LIN {X 0,Y 360.021,Z 1147.139,A -85,B 0,C 180,E1 17549.045,E2 17549.045} C_VEL
LIN {X 0,Y 360.007,Z 1146.189,A -85,B 0,C 180,E1 17546.018,E2 17546.018} C_VEL
LIN {X 0,Y 360.001,Z 1143.714,A -85,B 0,C 180,E1 17542.339,E2 17542.339} C_VEL
LIN {X 0,Y 360.288,Z 1139.777,A -85,B 0,C 180,E1 17538.798,E2 17538.798} C_VEL
LIN {X 0,Y 360.939,Z 1135.011,A -85,B 0,C 180,E1 17535.563,E2 17535.563} C_VEL
LIN {X 0,Y 362.46,Z 1127.574,A -85,B 0,C 180,E1 17531.617,E2 17531.617} C_VEL
LIN {X 0,Y 364.535,Z 1119.65,A -85,B 0,C 180,E1 17528.266,E2 17528.266} C_VEL
LIN {X 0,Y 367.67,Z 1109.706,A -85,B 0,C 180,E1 17524.725,E2 17524.725} C_VEL
LIN {X 0,Y 371.821,Z 1097.742,A -85,B 0,C 180,E1 17521.225,E2 17521.225} C_VEL
LIN {X 0,Y 376.526,Z 1085.225,A -85,B 0,C 180,E1 17518.099,E2 17518.099} C_VEL
LIN {X 0,Y 382.373,Z 1070.124,A -85,B 0,C 180,E1 17514.934,E2 17514.934} C_VEL
LIN {X 0,Y 388.351,Z 1054.921,A -85,B 0,C 180,E1 17512.209,E2 17512.209} C_VEL
LIN {X 0,Y 395.187,Z 1037.236,A -85,B 0,C 180,E1 17509.534,E2 17509.534} C_VEL
LIN {X 0,Y 401.308,Z 1020.991,A -85,B 0,C 180,E1 17507.432,E2 17507.432} C_VEL
LIN {X 0,Y 408.852,Z 999.928,A -85,B 0,C 180,E1 17505.125,E2 17505.125} C_VEL
LIN {X 0,Y 414.782,Z 982.18,A -85,B 0,C 180,E1 17503.481,E2 17503.481} C_VEL
LIN {X 0,Y 421.323,Z 961.181,A -85,B 0,C 180,E1 17501.824,E2 17501.824} C_VEL
LIN {X 0,Y 427.122,Z 940.304,A -85,B 0,C 180,E1 17500.463,E2 17500.463} C_VEL
LIN {X 0,Y 432.626,Z 918.319,A -85,B 0,C 180,E1 17499.262,E2 17499.262} C_VEL
LIN {X 0,Y 437.401,Z 895.765,A -85,B 0,C 180,E1 17498.28,E2 17498.28} C_VEL
LIN {X 0,Y 441.245,Z 874.481,A -85,B 0,C 180,E1 17497.536,E2 17497.536} C_VEL
LIN {X 0,Y 444.909,Z 848.294,A -85,B 0,C 180,E1 17496.842,E2 17496.842} C_VEL
LIN {X 0,Y 446.964,Z 825.929,A -85,B 0,C 180,E1 17496.396,E2 17496.396} C_VEL
LIN {X 0,Y 460.098,Z 603.079,A -85,B 0,C 180,E1 17492.792,E2 17492.792} C_VEL
LIN {X 0,Y 461.524,Z 577.948,A -85,B 0,C 180,E1 17492.371,E2 17492.371} C_VEL
LIN {X 0,Y 452.704,Z 561.651,A -85,B 0,C 180,E1 17490.201,E2 17490.201} C_VEL
LIN {X 0,Y 443.998,Z 546.554,A -85,B 0,C 180,E1 17487.859,E2 17487.859} C_VEL
LIN {X 0,Y 434.702,Z 531.507,A -85,B 0,C 180,E1 17485.075,E2 17485.075} C_VEL
LIN {X 0,Y 426.121,Z 518.593,A -85,B 0,C 180,E1 17482.16,E2 17482.16} C_VEL
LIN {X 0,Y 420.35,Z 510.714,A -85,B 0,C 180,E1 17479.959,E2 17479.959} C_VEL
LIN {X 0,Y 416.022,Z 505.286,A -85,B 0,C 180,E1 17478.135,E2 17478.135} C_VEL
LIN {X 0,Y 412.343,Z 500.609,A -85,B 0,C 180,E1 17476.41,E2 17476.41} C_VEL
LIN {X 0,Y 408.2,Z 495.981,A -85,B 0,C 180,E1 17474.251,E2 17474.251} C_VEL
LIN {X 0,Y 406.955,Z 494.027,A -85,B 0,C 180,E1 17473.498,E2 17473.498} C_VEL
LIN {X 0,Y 403.56,Z 490.738,A -85,B 0,C 180,E1 17471.36,E2 17471.36} C_VEL
LIN {X 0,Y 402.048,Z 488.022,A -85,B 0,C 180,E1 17470.17,E2 17470.17} C_VEL
LIN {X 0,Y 398.584,Z 485.25,A -85,B 0,C 180,E1 17467.206,E2 17467.206} C_VEL
LIN {X 0,Y 396.721,Z 481.774,A -85,B 0,C 180,E1 17464.771,E2 17464.771} C_VEL
LIN {X 0,Y 394.33,Z 480.47,A -85,B 0,C 180,E1 17458.838,E2 17458.838} C_VEL
LIN {X 0,Y 395.914,Z 481.333,A -85,B 0,C 180,E1 17452.891,E2 17452.891} C_VEL
LIN {X 0,Y 397.035,Z 482.238,A -85,B 0,C 180,E1 17451.236,E2 17451.236} C_VEL
LIN {X 0,Y 398.95,Z 485.758,A -85,B 0,C 180,E1 17448.873,E2 17448.873} C_VEL
LIN {X 0,Y 402.253,Z 488.401,A -85,B 0,C 180,E1 17446.121,E2 17446.121} C_VEL
LIN {X 0,Y 404.933,Z 492.456,A -85,B 0,C 180,E1 17444.166,E2 17444.166} C_VEL
LIN {X 0,Y 407.408,Z 494.631,A -85,B 0,C 180,E1 17442.692,E2 17442.692} C_VEL
LIN {X 0,Y 410.514,Z 498.843,A -85,B 0,C 180,E1 17440.95,E2 17440.95} C_VEL
LIN {X 0,Y 412.484,Z 500.879,A -85,B 0,C 180,E1 17439.977,E2 17439.977} C_VEL
LIN {X 0,Y 416.124,Z 505.413,A -85,B 0,C 180,E1 17438.282,E2 17438.282} C_VEL
LIN {X 0,Y 421.938,Z 512.849,A -85,B 0,C 180,E1 17435.871,E2 17435.871} C_VEL
LIN {X 0,Y 426.445,Z 518.715,A -85,B 0,C 180,E1 17434.197,E2 17434.197} C_VEL
LIN {X 0,Y 433.251,Z 527.659,A -85,B 0,C 180,E1 17431.913,E2 17431.913} C_VEL
LIN {X 0,Y 442.834,Z 541.129,A -85,B 0,C 180,E1 17429.053,E2 17429.053} C_VEL
LIN {X 0,Y 453.593,Z 557.288,A -85,B 0,C 180,E1 17426.215,E2 17426.215} C_VEL
LIN {X 0,Y 461.906,Z 570.817,A -85,B 0,C 180,E1 17424.222,E2 17424.222} C_VEL
LIN {X 0,Y 447.536,Z 809.905,A -85,B 0,C 180,E1 17420.364,E2 17420.364} C_VEL
LIN {X 0,Y 445.256,Z 833.988,A -85,B 0,C 180,E1 17419.851,E2 17419.851} C_VEL
LIN {X 0,Y 441.876,Z 857.908,A -85,B 0,C 180,E1 17419.139,E2 17419.139} C_VEL
LIN {X 0,Y 438.373,Z 878.069,A -85,B 0,C 180,E1 17418.381,E2 17418.381} C_VEL
LIN {X 0,Y 433.471,Z 901.517,A -85,B 0,C 180,E1 17417.281,E2 17417.281} C_VEL
LIN {X 0,Y 428.548,Z 921.582,A -85,B 0,C 180,E1 17416.134,E2 17416.134} C_VEL
LIN {X 0,Y 422.552,Z 943.344,A -85,B 0,C 180,E1 17414.652,E2 17414.652} C_VEL
LIN {X 0,Y 416.332,Z 963.34,A -85,B 0,C 180,E1 17413.006,E2 17413.006} C_VEL
LIN {X 0,Y 409.773,Z 982.956,A -85,B 0,C 180,E1 17411.118,E2 17411.118} C_VEL
LIN {X 0,Y 402.947,Z 1001.537,A -85,B 0,C 180,E1 17408.98,E2 17408.98} C_VEL
LIN {X 0,Y 396.645,Z 1018.01,A -85,B 0,C 180,E1 17406.778,E2 17406.778} C_VEL
LIN {X 0,Y 389.979,Z 1034.602,A -85,B 0,C 180,E1 17404.16,E2 17404.16} C_VEL
LIN {X 0,Y 384.496,Z 1048.038,A -85,B 0,C 180,E1 17401.689,E2 17401.689} C_VEL
LIN {X 0,Y 378.3,Z 1063.208,A -85,B 0,C 180,E1 17398.409,E2 17398.409} C_VEL
LIN {X 0,Y 373.754,Z 1074.487,A -85,B 0,C 180,E1 17395.513,E2 17395.513} C_VEL
LIN {X 0,Y 369.423,Z 1085.843,A -85,B 0,C 180,E1 17392.1,E2 17392.1} C_VEL
LIN {X 0,Y 365.952,Z 1095.521,A -85,B 0,C 180,E1 17388.538,E2 17388.538} C_VEL
LIN {X 0,Y 363.364,Z 1103.901,A -85,B 0,C 180,E1 17384.828,E2 17384.828} C_VEL
LIN {X 0,Y 361.661,Z 1110.331,A -85,B 0,C 180,E1 17381.159,E2 17381.159} C_VEL
LIN {X 0,Y 360.74,Z 1114.959,A -85,B 0,C 180,E1 17377.806,E2 17377.806} C_VEL
LIN {X 0,Y 360.203,Z 1118.85,A -85,B 0,C 180,E1 17373.82,E2 17373.82} C_VEL
LIN {X 0,Y 360.063,Z 1120.727,A -85,B 0,C 180,E1 17370.636,E2 17370.636} C_VEL
LIN {X 0,Y 360.023,Z 1121.58,A -85,B 0,C 180,E1 17367.453,E2 17367.453} C_VEL
LIN {X 0,Y 360.077,Z 1121.318,A -85,B 0,C 180,E1 17363.783,E2 17363.783} C_VEL
LIN {X 0,Y 360.228,Z 1119.57,A -85,B 0,C 180,E1 17360.192,E2 17360.192} C_VEL
LIN {X 0,Y 360.632,Z 1116.98,A -85,B 0,C 180,E1 17357.022,E2 17357.022} C_VEL
LIN {X 0,Y 361.666,Z 1112.414,A -85,B 0,C 180,E1 17353.124,E2 17353.124} C_VEL
LIN {X 0,Y 363.294,Z 1106.604,A -85,B 0,C 180,E1 17349.541,E2 17349.541} C_VEL
LIN {X 0,Y 365.631,Z 1099.754,A -85,B 0,C 180,E1 17346.125,E2 17346.125} C_VEL
LIN {X 0,Y 369.351,Z 1090.062,A -85,B 0,C 180,E1 17342.249,E2 17342.249} C_VEL
LIN {X 0,Y 373.414,Z 1080.418,A -85,B 0,C 180,E1 17339.061,E2 17339.061} C_VEL
LIN {X 0,Y 379.154,Z 1067.334,A -85,B 0,C 180,E1 17335.459,E2 17335.459} C_VEL
LIN {X 0,Y 382.472,Z 1059.991,A -85,B 0,C 180,E1 17333.7,E2 17333.7} C_VEL
LIN {X 0,Y 383.453,Z 1055.951,A -85,B 0,C 180,E1 17332.718,E2 17332.718} C_VEL
LIN {X 0,Y 383.271,Z 1045.58,A -85,B 0,C 180,E1 17329.947,E2 17329.947} C_VEL
LIN {X 0,Y 384.403,Z 1041.717,A -85,B 0,C 180,E1 17329.157,E2 17329.157} C_VEL
LIN {X 0,Y 391.561,Z 1025.886,A -85,B 0,C 180,E1 17326.488,E2 17326.488} C_VEL
LIN {X 0,Y 399.116,Z 1008.809,A -85,B 0,C 180,E1 17324.027,E2 17324.027} C_VEL
LIN {X 0,Y 406.608,Z 990.541,A -85,B 0,C 180,E1 17321.831,E2 17321.831} C_VEL
LIN {X 0,Y 413.61,Z 972.484,A -85,B 0,C 180,E1 17319.973,E2 17319.973} C_VEL
LIN {X 0,Y 420.966,Z 951.548,A -85,B 0,C 180,E1 17318.168,E2 17318.168} C_VEL
LIN {X 0,Y 426.659,Z 933.743,A -85,B 0,C 180,E1 17316.866,E2 17316.866} C_VEL
LIN {X 0,Y 432.999,Z 911.71,A -85,B 0,C 180,E1 17315.511,E2 17315.511} C_VEL
LIN {X 0,Y 438.107,Z 890.792,A -85,B 0,C 180,E1 17314.453,E2 17314.453} C_VEL
LIN {X 0,Y 443.011,Z 867.537,A -85,B 0,C 180,E1 17313.49,E2 17313.49} C_VEL
LIN {X 0,Y 446.93,Z 843.553,A -85,B 0,C 180,E1 17312.732,E2 17312.732} C_VEL
LIN {X 0,Y 449.974,Z 819.403,A -85,B 0,C 180,E1 17312.153,E2 17312.153} C_VEL
LIN {X 0,Y 453.059,Z 776.212,A -85,B 0,C 180,E1 17311.426,E2 17311.426} C_VEL
LIN {X 0,Y 465.941,Z 580.402,A -85,B 0,C 180,E1 17308.294,E2 17308.294} C_VEL
LIN {X 0,Y 456.566,Z 565.613,A -85,B 0,C 180,E1 17305.663,E2 17305.663} C_VEL
LIN {X 0,Y 448.896,Z 554.256,A -85,B 0,C 180,E1 17303.255,E2 17303.255} C_VEL
LIN {X 0,Y 442.446,Z 545.251,A -85,B 0,C 180,E1 17300.99,E2 17300.99} C_VEL
LIN {X 0,Y 436.973,Z 537.664,A -85,B 0,C 180,E1 17298.823,E2 17298.823} C_VEL
LIN {X 0,Y 432.55,Z 531.917,A -85,B 0,C 180,E1 17296.865,E2 17296.865} C_VEL
LIN {X 0,Y 428.948,Z 527.145,A -85,B 0,C 180,E1 17295.065,E2 17295.065} C_VEL
LIN {X 0,Y 425.508,Z 522.542,A -85,B 0,C 180,E1 17293.107,E2 17293.107} C_VEL
LIN {X 0,Y 421.619,Z 518.027,A -85,B 0,C 180,E1 17290.522,E2 17290.522} C_VEL
LIN {X 0,Y 420.468,Z 516.135,A -85,B 0,C 180,E1 17289.582,E2 17289.582} C_VEL
LIN {X 0,Y 417.506,Z 513.236,A -85,B 0,C 180,E1 17286.877,E2 17286.877} C_VEL
LIN {X 0,Y 416.111,Z 510.251,A -85,B 0,C 180,E1 17284.963,E2 17284.963} C_VEL
LIN {X 0,Y 413.805,Z 508.946,A -85,B 0,C 180,E1 17278.615,E2 17278.615} C_VEL
LIN {X 0,Y 416.185,Z 510.264,A -85,B 0,C 180,E1 17272.407,E2 17272.407} C_VEL
LIN {X 0,Y 418.1,Z 514.063,A -85,B 0,C 180,E1 17269.946,E2 17269.946} C_VEL
LIN {X 0,Y 420.981,Z 516.748,A -85,B 0,C 180,E1 17267.472,E2 17267.472} C_VEL
LIN {X 0,Y 423.84,Z 520.88,A -85,B 0,C 180,E1 17265.379,E2 17265.379} C_VEL
LIN {X 0,Y 425.556,Z 522.658,A -85,B 0,C 180,E1 17264.323,E2 17264.323} C_VEL
LIN {X 0,Y 429.149,Z 527.301,A -85,B 0,C 180,E1 17262.298,E2 17262.298} C_VEL
LIN {X 0,Y 434.821,Z 535.328,A -85,B 0,C 180,E1 17259.541,E2 17259.541} C_VEL
LIN {X 0,Y 442.077,Z 546.499,A -85,B 0,C 180,E1 17256.542,E2 17256.542} C_VEL
LIN {X 0,Y 450.552,Z 560.198,A -85,B 0,C 180,E1 17253.543,E2 17253.543} C_VEL
LIN {X 0,Y 459.042,Z 574.94,A -85,B 0,C 180,E1 17250.903,E2 17250.903} C_VEL
LIN {X 0,Y 465.746,Z 587.338,A -85,B 0,C 180,E1 17249.008,E2 17249.008} C_VEL
LIN {X 0,Y 451.666,Z 802.695,A -85,B 0,C 180,E1 17245.552,E2 17245.552} C_VEL
LIN {X 0,Y 448.973,Z 838.695,A -85,B 0,C 180,E1 17244.934,E2 17244.934} C_VEL
LIN {X 0,Y 445.869,Z 862.066,A -85,B 0,C 180,E1 17244.4,E2 17244.4} C_VEL
LIN {X 0,Y 441.598,Z 886.506,A -85,B 0,C 180,E1 17243.673,E2 17243.673} C_VEL
LIN {X 0,Y 436.736,Z 908.538,A -85,B 0,C 180,E1 17242.813,E2 17242.813} C_VEL
LIN {X 0,Y 431.378,Z 929.766,A -85,B 0,C 180,E1 17241.792,E2 17241.792} C_VEL
LIN {X 0,Y 424.687,Z 952.666,A -85,B 0,C 180,E1 17240.432,E2 17240.432} C_VEL
LIN {X 0,Y 418.351,Z 972.088,A -85,B 0,C 180,E1 17239.049,E2 17239.049} C_VEL
LIN {X 0,Y 410.452,Z 994.126,A -85,B 0,C 180,E1 17237.16,E2 17237.16} C_VEL
LIN {X 0,Y 403.498,Z 1012.027,A -85,B 0,C 180,E1 17235.333,E2 17235.333} C_VEL
LIN {X 0,Y 395.194,Z 1032.173,A -85,B 0,C 180,E1 17232.891,E2 17232.891} C_VEL
LIN {X 0,Y 388.422,Z 1047.829,A -85,B 0,C 180,E1 17230.639,E2 17230.639} C_VEL
LIN {X 0,Y 381.089,Z 1064.48,A -85,B 0,C 180,E1 17227.837,E2 17227.837} C_VEL
LIN {X 0,Y 374.702,Z 1078.671,A -85,B 0,C 180,E1 17224.992,E2 17224.992} C_VEL
LIN {X 0,Y 368.65,Z 1092.528,A -85,B 0,C 180,E1 17221.748,E2 17221.748} C_VEL
LIN {X 0,Y 363.38,Z 1104.882,A -85,B 0,C 180,E1 17218.248,E2 17218.248} C_VEL
LIN {X 0,Y 359.256,Z 1115.568,A -85,B 0,C 180,E1 17214.676,E2 17214.676} C_VEL
LIN {X 0,Y 356.061,Z 1124.76,A -85,B 0,C 180,E1 17210.894,E2 17210.894} C_VEL
LIN {X 0,Y 354.027,Z 1131.913,A -85,B 0,C 180,E1 17207.325,E2 17207.325} C_VEL
LIN {X 0,Y 352.669,Z 1138.254,A -85,B 0,C 180,E1 17203.277,E2 17203.277} C_VEL
LIN {X 0,Y 352.135,Z 1142.289,A -85,B 0,C 180,E1 17199.809,E2 17199.809} C_VEL
LIN {X 0,Y 351.99,Z 1145.232,A -85,B 0,C 180,E1 17196.197,E2 17196.197} C_VEL
LIN {X 0,Y 352.005,Z 1146.752,A -85,B 0,C 180,E1 17192.442,E2 17192.442} C_VEL
LIN {X 0,Y 352.021,Z 1146.896,A -85,B 0,C 180,E1 17189.349,E2 17189.349} C_VEL
LIN {X 0,Y 352.01,Z 1146.032,A -85,B 0,C 180,E1 17186.254,E2 17186.254} C_VEL
LIN {X 0,Y 352.007,Z 1143.92,A -85,B 0,C 180,E1 17182.82,E2 17182.82} C_VEL
LIN {X 0,Y 352.277,Z 1139.878,A -85,B 0,C 180,E1 17178.872,E2 17178.872} C_VEL
LIN {X 0,Y 352.933,Z 1135.2,A -85,B 0,C 180,E1 17175.563,E2 17175.563} C_VEL
LIN {X 0,Y 354.375,Z 1128.395,A -85,B 0,C 180,E1 17171.748,E2 17171.748} C_VEL
LIN {X 0,Y 356.738,Z 1119.698,A -85,B 0,C 180,E1 17167.939,E2 17167.939} C_VEL
LIN {X 0,Y 359.833,Z 1110.269,A -85,B 0,C 180,E1 17164.487,E2 17164.487} C_VEL
LIN {X 0,Y 364.275,Z 1098.066,A -85,B 0,C 180,E1 17160.795,E2 17160.795} C_VEL
LIN {X 0,Y 368.944,Z 1086.11,A -85,B 0,C 180,E1 17157.731,E2 17157.731} C_VEL
LIN {X 0,Y 375.269,Z 1070.472,A -85,B 0,C 180,E1 17154.357,E2 17154.357} C_VEL
LIN {X 0,Y 381.092,Z 1056.192,A -85,B 0,C 180,E1 17151.742,E2 17151.742} C_VEL
LIN {X 0,Y 388.512,Z 1037.782,A -85,B 0,C 180,E1 17148.885,E2 17148.885} C_VEL
LIN {X 0,Y 394.815,Z 1021.615,A -85,B 0,C 180,E1 17146.76,E2 17146.76} C_VEL
LIN {X 0,Y 402.339,Z 1001.417,A -85,B 0,C 180,E1 17144.5,E2 17144.5} C_VEL
LIN {X 0,Y 408.661,Z 983.099,A -85,B 0,C 180,E1 17142.775,E2 17142.775} C_VEL
LIN {X 0,Y 415.374,Z 962.357,A -85,B 0,C 180,E1 17141.109,E2 17141.109} C_VEL
LIN {X 0,Y 421.585,Z 940.65,A -85,B 0,C 180,E1 17139.679,E2 17139.679} C_VEL
LIN {X 0,Y 426.673,Z 920.918,A -85,B 0,C 180,E1 17138.587,E2 17138.587} C_VEL
LIN {X 0,Y 432.034,Z 896.834,A -85,B 0,C 180,E1 17137.509,E2 17137.509} C_VEL
LIN {X 0,Y 435.953,Z 875.808,A -85,B 0,C 180,E1 17136.764,E2 17136.764} C_VEL
LIN {X 0,Y 439.748,Z 850.119,A -85,B 0,C 180,E1 17136.067,E2 17136.067} C_VEL
LIN {X 0,Y 441.958,Z 827.356,A -85,B 0,C 180,E1 17135.604,E2 17135.604} C_VEL
LIN {X 0,Y 455.463,Z 605.528,A -85,B 0,C 180,E1 17131.999,E2 17131.999} C_VEL
LIN {X 0,Y 456.828,Z 581.647,A -85,B 0,C 180,E1 17131.591,E2 17131.591} C_VEL
LIN {X 0,Y 448.666,Z 566.477,A -85,B 0,C 180,E1 17129.506,E2 17129.506} C_VEL
LIN {X 0,Y 440.17,Z 551.554,A -85,B 0,C 180,E1 17127.131,E2 17127.131} C_VEL
LIN {X 0,Y 431.21,Z 536.958,A -85,B 0,C 180,E1 17124.341,E2 17124.341} C_VEL
LIN {X 0,Y 423.645,Z 525.381,A -85,B 0,C 180,E1 17121.677,E2 17121.677} C_VEL
LIN {X 0,Y 418.4,Z 518.079,A -85,B 0,C 180,E1 17119.619,E2 17119.619} C_VEL
LIN {X 0,Y 413.999,Z 512.534,A -85,B 0,C 180,E1 17117.717,E2 17117.717} C_VEL
LIN {X 0,Y 409.872,Z 507.315,A -85,B 0,C 180,E1 17115.711,E2 17115.711} C_VEL
LIN {X 0,Y 406.508,Z 503.334,A -85,B 0,C 180,E1 17113.876,E2 17113.876} C_VEL
LIN {X 0,Y 405.511,Z 501.749,A -85,B 0,C 180,E1 17113.257,E2 17113.257} C_VEL
LIN {X 0,Y 402.185,Z 498.42,A -85,B 0,C 180,E1 17111.109,E2 17111.109} C_VEL
LIN {X 0,Y 400.699,Z 495.801,A -85,B 0,C 180,E1 17109.915,E2 17109.915} C_VEL
LIN {X 0,Y 397.338,Z 492.954,A -85,B 0,C 180,E1 17106.938,E2 17106.938} C_VEL
LIN {X 0,Y 395.643,Z 489.657,A -85,B 0,C 180,E1 17104.639,E2 17104.639} C_VEL
LIN {X 0,Y 393.346,Z 488.404,A -85,B 0,C 180,E1 17098.689,E2 17098.689} C_VEL
LIN {X 0,Y 395.126,Z 489.357,A -85,B 0,C 180,E1 17092.585,E2 17092.585} C_VEL
LIN {X 0,Y 395.949,Z 490.184,A -85,B 0,C 180,E1 17091.358,E2 17091.358} C_VEL
LIN {X 0,Y 397.838,Z 493.644,A -85,B 0,C 180,E1 17088.988,E2 17088.988} C_VEL
LIN {X 0,Y 400.915,Z 496.143,A -85,B 0,C 180,E1 17086.368,E2 17086.368} C_VEL
LIN {X 0,Y 403.648,Z 500.266,A -85,B 0,C 180,E1 17084.335,E2 17084.335} C_VEL
LIN {X 0,Y 405.917,Z 502.32,A -85,B 0,C 180,E1 17082.954,E2 17082.954} C_VEL
LIN {X 0,Y 409.163,Z 506.667,A -85,B 0,C 180,E1 17081.107,E2 17081.107} C_VEL
LIN {X 0,Y 410.896,Z 508.579,A -85,B 0,C 180,E1 17080.23,E2 17080.23} C_VEL
LIN {X 0,Y 414.721,Z 513.249,A -85,B 0,C 180,E1 17078.427,E2 17078.427} C_VEL
LIN {X 0,Y 420.302,Z 520.698,A -85,B 0,C 180,E1 17076.07,E2 17076.07} C_VEL
LIN {X 0,Y 424.366,Z 526.044,A -85,B 0,C 180,E1 17074.532,E2 17074.532} C_VEL
LIN {X 0,Y 431.029,Z 534.977,A -85,B 0,C 180,E1 17072.245,E2 17072.245} C_VEL
LIN {X 0,Y 440.173,Z 548.038,A -85,B 0,C 180,E1 17069.451,E2 17069.451} C_VEL
LIN {X 0,Y 450.55,Z 563.877,A -85,B 0,C 180,E1 17066.645,E2 17066.645} C_VEL
LIN {X 0,Y 457.223,Z 575.002,A -85,B 0,C 180,E1 17064.988,E2 17064.988} C_VEL
LIN {X 0,Y 442.604,Z 810.925,A -85,B 0,C 180,E1 17061.167,E2 17061.167} C_VEL
LIN {X 0,Y 440.169,Z 835.453,A -85,B 0,C 180,E1 17060.636,E2 17060.636} C_VEL
LIN {X 0,Y 436.755,Z 858.824,A -85,B 0,C 180,E1 17059.932,E2 17059.932} C_VEL
LIN {X 0,Y 432.87,Z 880.499,A -85,B 0,C 180,E1 17059.106,E2 17059.106} C_VEL
LIN {X 0,Y 427.839,Z 903.446,A -85,B 0,C 180,E1 17058.004,E2 17058.004} C_VEL
LIN {X 0,Y 422.801,Z 923.327,A -85,B 0,C 180,E1 17056.851,E2 17056.851} C_VEL
LIN {X 0,Y 416.264,Z 946.02,A -85,B 0,C 180,E1 17055.267,E2 17055.267} C_VEL
LIN {X 0,Y 410.312,Z 964.555,A -85,B 0,C 180,E1 17053.717,E2 17053.717} C_VEL
LIN {X 0,Y 403.26,Z 984.833,A -85,B 0,C 180,E1 17051.726,E2 17051.726} C_VEL
LIN {X 0,Y 396.718,Z 1002.088,A -85,B 0,C 180,E1 17049.712,E2 17049.712} C_VEL
LIN {X 0,Y 389.738,Z 1019.754,A -85,B 0,C 180,E1 17047.314,E2 17047.314} C_VEL
LIN {X 0,Y 382.826,Z 1036.229,A -85,B 0,C 180,E1 17044.64,E2 17044.64} C_VEL
LIN {X 0,Y 376.399,Z 1051.526,A -85,B 0,C 180,E1 17041.734,E2 17041.734} C_VEL
LIN {X 0,Y 370.38,Z 1065.511,A -85,B 0,C 180,E1 17038.544,E2 17038.544} C_VEL
LIN {X 0,Y 365.346,Z 1077.712,A -85,B 0,C 180,E1 17035.274,E2 17035.274} C_VEL
LIN {X 0,Y 361.017,Z 1088.476,A -85,B 0,C 180,E1 17031.786,E2 17031.786} C_VEL
LIN {X 0,Y 357.828,Z 1097.232,A -85,B 0,C 180,E1 17028.407,E2 17028.407} C_VEL
LIN {X 0,Y 355.095,Z 1105.735,A -85,B 0,C 180,E1 17024.347,E2 17024.347} C_VEL
LIN {X 0,Y 353.596,Z 1111.42,A -85,B 0,C 180,E1 17020.921,E2 17020.921} C_VEL
LIN {X 0,Y 352.608,Z 1116.414,A -85,B 0,C 180,E1 17017.004,E2 17017.004} C_VEL
LIN {X 0,Y 352.186,Z 1119.493,A -85,B 0,C 180,E1 17013.418,E2 17013.418} C_VEL
LIN {X 0,Y 352.082,Z 1121.227,A -85,B 0,C 180,E1 17010.163,E2 17010.163} C_VEL
LIN {X 0,Y 352.03,Z 1121.965,A -85,B 0,C 180,E1 17006.254,E2 17006.254} C_VEL
LIN {X 0,Y 352.083,Z 1121.26,A -85,B 0,C 180,E1 17002.822,E2 17002.822} C_VEL
LIN {X 0,Y 352.284,Z 1119.651,A -85,B 0,C 180,E1 16999.699,E2 16999.699} C_VEL
LIN {X 0,Y 352.803,Z 1116.766,A -85,B 0,C 180,E1 16996.227,E2 16996.227} C_VEL
LIN {X 0,Y 354.071,Z 1111.648,A -85,B 0,C 180,E1 16992.072,E2 16992.072} C_VEL
LIN {X 0,Y 355.774,Z 1106.228,A -85,B 0,C 180,E1 16988.743,E2 16988.743} C_VEL
LIN {X 0,Y 358.654,Z 1098.527,A -85,B 0,C 180,E1 16984.928,E2 16984.928} C_VEL
LIN {X 0,Y 362.407,Z 1089.336,A -85,B 0,C 180,E1 16981.31,E2 16981.31} C_VEL
LIN {X 0,Y 367.26,Z 1078.544,A -85,B 0,C 180,E1 16977.749,E2 16977.749} C_VEL
LIN {X 0,Y 372.906,Z 1066.213,A -85,B 0,C 180,E1 16974.419,E2 16974.419} C_VEL
LIN {X 0,Y 379.387,Z 1052.505,A -85,B 0,C 180,E1 16971.272,E2 16971.272} C_VEL
LIN {X 0,Y 384.403,Z 1041.717,A -85,B 0,C 180,E1 16969.157,E2 16969.157} C_VEL
LIN {X 0,Y 385.668,Z 1037.2,A -85,B 0,C 180,E1 16968.245,E2 16968.245} C_VEL
LIN {X 0,Y 386.299,Z 1026.065,A -85,B 0,C 180,E1 16965.758,E2 16965.758} C_VEL
LIN {X 0,Y 387.885,Z 1021.15,A -85,B 0,C 180,E1 16964.892,E2 16964.892} C_VEL
LIN {X 0,Y 395.765,Z 1003.299,A -85,B 0,C 180,E1 16962.461,E2 16962.461} C_VEL
LIN {X 0,Y 403.184,Z 985.67,A -85,B 0,C 180,E1 16960.416,E2 16960.416} C_VEL
LIN {X 0,Y 411.026,Z 965.256,A -85,B 0,C 180,E1 16958.434,E2 16958.434} C_VEL
LIN {X 0,Y 417.619,Z 946.566,A -85,B 0,C 180,E1 16956.9,E2 16956.9} C_VEL
LIN {X 0,Y 424.83,Z 923.651,A -85,B 0,C 180,E1 16955.337,E2 16955.337} C_VEL
LIN {X 0,Y 430.385,Z 903.505,A -85,B 0,C 180,E1 16954.2,E2 16954.2} C_VEL
LIN {X 0,Y 436.159,Z 878.888,A -85,B 0,C 180,E1 16953.067,E2 16953.067} C_VEL
LIN {X 0,Y 440.155,Z 858.208,A -85,B 0,C 180,E1 16952.313,E2 16952.313} C_VEL
LIN {X 0,Y 443.857,Z 834.378,A -85,B 0,C 180,E1 16951.629,E2 16951.629} C_VEL
LIN {X 0,Y 446.34,Z 810.78,A -85,B 0,C 180,E1 16951.137,E2 16951.137} C_VEL
LIN {X 0,Y 461.735,Z 584.813,A -85,B 0,C 180,E1 16947.505,E2 16947.505} C_VEL
LIN {X 0,Y 453.04,Z 571.066,A -85,B 0,C 180,E1 16944.968,E2 16944.968} C_VEL
LIN {X 0,Y 445.602,Z 559.758,A -85,B 0,C 180,E1 16942.529,E2 16942.529} C_VEL
LIN {X 0,Y 437.632,Z 548.625,A -85,B 0,C 180,E1 16939.556,E2 16939.556} C_VEL
LIN {X 0,Y 434.06,Z 543.78,A -85,B 0,C 180,E1 16938.049,E2 16938.049} C_VEL
LIN {X 0,Y 430.752,Z 539.299,A -85,B 0,C 180,E1 16936.52,E2 16936.52} C_VEL
LIN {X 0,Y 427.227,Z 534.581,A -85,B 0,C 180,E1 16934.711,E2 16934.711} C_VEL
LIN {X 0,Y 423.562,Z 529.609,A -85,B 0,C 180,E1 16932.544,E2 16932.544} C_VEL
LIN {X 0,Y 420.367,Z 525.859,A -85,B 0,C 180,E1 16930.346,E2 16930.346} C_VEL
LIN {X 0,Y 419.325,Z 524.012,A -85,B 0,C 180,E1 16929.47,E2 16929.47} C_VEL
LIN {X 0,Y 416.403,Z 521.127,A -85,B 0,C 180,E1 16926.757,E2 16926.757} C_VEL
LIN {X 0,Y 414.936,Z 518.11,A -85,B 0,C 180,E1 16924.7,E2 16924.7} C_VEL
LIN {X 0,Y 412.83,Z 516.887,A -85,B 0,C 180,E1 16918.612,E2 16918.612} C_VEL
LIN {X 0,Y 415.11,Z 518.196,A -85,B 0,C 180,E1 16912.526,E2 16912.526} C_VEL
LIN {X 0,Y 416.993,Z 521.95,A -85,B 0,C 180,E1 16910.058,E2 16910.058} C_VEL
LIN {X 0,Y 419.694,Z 524.519,A -85,B 0,C 180,E1 16907.688,E2 16907.688} C_VEL
LIN {X 0,Y 422.67,Z 528.784,A -85,B 0,C 180,E1 16905.477,E2 16905.477} C_VEL
LIN {X 0,Y 424.144,Z 530.395,A -85,B 0,C 180,E1 16904.55,E2 16904.55} C_VEL
LIN {X 0,Y 428.654,Z 536.433,A -85,B 0,C 180,E1 16901.997,E2 16901.997} C_VEL
LIN {X 0,Y 433.667,Z 543.917,A -85,B 0,C 180,E1 16899.555,E2 16899.555} C_VEL
LIN {X 0,Y 439.634,Z 553.146,A -85,B 0,C 180,E1 16897.042,E2 16897.042} C_VEL
LIN {X 0,Y 447.827,Z 566.642,A -85,B 0,C 180,E1 16894.048,E2 16894.048} C_VEL
LIN {X 0,Y 456.142,Z 581.34,A -85,B 0,C 180,E1 16891.382,E2 16891.382} C_VEL
LIN {X 0,Y 461.509,Z 591.612,A -85,B 0,C 180,E1 16889.803,E2 16889.803} C_VEL
LIN {X 0,Y 446.895,Z 809.021,A -85,B 0,C 180,E1 16886.308,E2 16886.308} C_VEL
LIN {X 0,Y 444.175,Z 841.594,A -85,B 0,C 180,E1 16885.729,E2 16885.729} C_VEL
LIN {X 0,Y 441.087,Z 863.761,A -85,B 0,C 180,E1 16885.212,E2 16885.212} C_VEL
LIN {X 0,Y 436.208,Z 889.98,A -85,B 0,C 180,E1 16884.402,E2 16884.402} C_VEL
LIN {X 0,Y 431.501,Z 910.517,A -85,B 0,C 180,E1 16883.584,E2 16883.584} C_VEL
LIN {X 0,Y 425.236,Z 934.148,A -85,B 0,C 180,E1 16882.412,E2 16882.412} C_VEL
LIN {X 0,Y 418.761,Z 955.26,A -85,B 0,C 180,E1 16881.115,E2 16881.115} C_VEL
LIN {X 0,Y 411.418,Z 976.877,A -85,B 0,C 180,E1 16879.526,E2 16879.526} C_VEL
LIN {X 0,Y 403.902,Z 996.765,A -85,B 0,C 180,E1 16877.749,E2 16877.749} C_VEL
LIN {X 0,Y 396.077,Z 1016.226,A -85,B 0,C 180,E1 16875.7,E2 16875.7} C_VEL
LIN {X 0,Y 388.082,Z 1034.617,A -85,B 0,C 180,E1 16873.365,E2 16873.365} C_VEL
LIN {X 0,Y 380.377,Z 1051.862,A -85,B 0,C 180,E1 16870.794,E2 16870.794} C_VEL
LIN {X 0,Y 372.817,Z 1068.052,A -85,B 0,C 180,E1 16867.892,E2 16867.892} C_VEL
LIN {X 0,Y 366.369,Z 1081.972,A -85,B 0,C 180,E1 16864.969,E2 16864.969} C_VEL
LIN {X 0,Y 359.996,Z 1095.834,A -85,B 0,C 180,E1 16861.478,E2 16861.478} C_VEL
LIN {X 0,Y 355.009,Z 1107.294,A -85,B 0,C 180,E1 16858.058,E2 16858.058} C_VEL
LIN {X 0,Y 350.655,Z 1118.085,A -85,B 0,C 180,E1 16854.149,E2 16854.149} C_VEL
LIN {X 0,Y 347.892,Z 1125.974,A -85,B 0,C 180,E1 16850.703,E2 16850.703} C_VEL
LIN {X 0,Y 345.578,Z 1134.05,A -85,B 0,C 180,E1 16846.3,E2 16846.3} C_VEL
LIN {X 0,Y 344.562,Z 1138.961,A -85,B 0,C 180,E1 16842.826,E2 16842.826} C_VEL
LIN {X 0,Y 344.071,Z 1143.02,A -85,B 0,C 180,E1 16839.029,E2 16839.029} C_VEL
LIN {X 0,Y 343.973,Z 1145.547,A -85,B 0,C 180,E1 16835.17,E2 16835.17} C_VEL
LIN {X 0,Y 344.024,Z 1146.545,A -85,B 0,C 180,E1 16831.999,E2 16831.999} C_VEL
LIN {X 0,Y 344.034,Z 1146.539,A -85,B 0,C 180,E1 16828.834,E2 16828.834} C_VEL
LIN {X 0,Y 343.996,Z 1145.383,A -85,B 0,C 180,E1 16825.332,E2 16825.332} C_VEL
LIN {X 0,Y 344.059,Z 1142.591,A -85,B 0,C 180,E1 16821.477,E2 16821.477} C_VEL
LIN {X 0,Y 344.377,Z 1138.896,A -85,B 0,C 180,E1 16818.091,E2 16818.091} C_VEL
LIN {X 0,Y 345.219,Z 1133.811,A -85,B 0,C 180,E1 16814.546,E2 16814.546} C_VEL
LIN {X 0,Y 347.068,Z 1126.096,A -85,B 0,C 180,E1 16810.404,E2 16810.404} C_VEL
LIN {X 0,Y 349.499,Z 1118.08,A -85,B 0,C 180,E1 16806.924,E2 16806.924} C_VEL
LIN {X 0,Y 353.476,Z 1106.855,A -85,B 0,C 180,E1 16802.907,E2 16802.907} C_VEL
LIN {X 0,Y 357.553,Z 1096.347,A -85,B 0,C 180,E1 16799.777,E2 16799.777} C_VEL
LIN {X 0,Y 363.074,Z 1083.054,A -85,B 0,C 180,E1 16796.389,E2 16796.389} C_VEL
LIN {X 0,Y 369.196,Z 1068.441,A -85,B 0,C 180,E1 16793.289,E2 16793.289} C_VEL
LIN {X 0,Y 376.122,Z 1052.258,A -85,B 0,C 180,E1 16790.355,E2 16790.355} C_VEL
LIN {X 0,Y 383.149,Z 1035.228,A -85,B 0,C 180,E1 16787.779,E2 16787.779} C_VEL
LIN {X 0,Y 390.094,Z 1017.992,A -85,B 0,C 180,E1 16785.539,E2 16785.539} C_VEL
LIN {X 0,Y 397.569,Z 998.152,A -85,B 0,C 180,E1 16783.378,E2 16783.378} C_VEL
LIN {X 0,Y 404.148,Z 979.541,A -85,B 0,C 180,E1 16781.654,E2 16781.654} C_VEL
LIN {X 0,Y 411.479,Z 956.84,A -85,B 0,C 180,E1 16779.905,E2 16779.905} C_VEL
LIN {X 0,Y 417.259,Z 936.915,A -85,B 0,C 180,E1 16778.629,E2 16778.629} C_VEL
LIN {X 0,Y 423.513,Z 912.305,A -85,B 0,C 180,E1 16777.341,E2 16777.341} C_VEL
LIN {X 0,Y 428.05,Z 891.488,A -85,B 0,C 180,E1 16776.472,E2 16776.472} C_VEL
LIN {X 0,Y 432.473,Z 867.086,A -85,B 0,C 180,E1 16775.669,E2 16775.669} C_VEL
LIN {X 0,Y 435.556,Z 844.232,A -85,B 0,C 180,E1 16775.103,E2 16775.103} C_VEL
LIN {X 0,Y 437.815,Z 818.435,A -85,B 0,C 180,E1 16774.61,E2 16774.61} C_VEL
LIN {X 0,Y 451.553,Z 598.009,A -85,B 0,C 180,E1 16771.029,E2 16771.029} C_VEL
LIN {X 0,Y 452.244,Z 585.498,A -85,B 0,C 180,E1 16770.805,E2 16770.805} C_VEL
LIN {X 0,Y 443.341,Z 568.684,A -85,B 0,C 180,E1 16768.417,E2 16768.417} C_VEL
LIN {X 0,Y 434.544,Z 553.46,A -85,B 0,C 180,E1 16765.815,E2 16765.815} C_VEL
LIN {X 0,Y 426.89,Z 540.961,A -85,B 0,C 180,E1 16763.282,E2 16763.282} C_VEL
LIN {X 0,Y 419.163,Z 529.088,A -85,B 0,C 180,E1 16760.382,E2 16760.382} C_VEL
LIN {X 0,Y 415.836,Z 524.734,A -85,B 0,C 180,E1 16759.015,E2 16759.015} C_VEL
LIN {X 0,Y 412.292,Z 520.071,A -85,B 0,C 180,E1 16757.428,E2 16757.428} C_VEL
LIN {X 0,Y 408.234,Z 514.884,A -85,B 0,C 180,E1 16755.412,E2 16755.412} C_VEL
LIN {X 0,Y 404.833,Z 510.687,A -85,B 0,C 180,E1 16753.498,E2 16753.498} C_VEL
LIN {X 0,Y 403.842,Z 509.301,A -85,B 0,C 180,E1 16752.876,E2 16752.876} C_VEL
LIN {X 0,Y 400.546,Z 505.671,A -85,B 0,C 180,E1 16750.645,E2 16750.645} C_VEL
LIN {X 0,Y 399.358,Z 503.575,A -85,B 0,C 180,E1 16749.657,E2 16749.657} C_VEL
LIN {X 0,Y 396.102,Z 500.657,A -85,B 0,C 180,E1 16746.668,E2 16746.668} C_VEL
LIN {X 0,Y 394.567,Z 497.541,A -85,B 0,C 180,E1 16744.506,E2 16744.506} C_VEL
LIN {X 0,Y 392.361,Z 496.333,A -85,B 0,C 180,E1 16738.394,E2 16738.394} C_VEL
LIN {X 0,Y 394.448,Z 497.435,A -85,B 0,C 180,E1 16732.132,E2 16732.132} C_VEL
LIN {X 0,Y 395.09,Z 498.761,A -85,B 0,C 180,E1 16731.119,E2 16731.119} C_VEL
LIN {X 0,Y 397.309,Z 502.112,A -85,B 0,C 180,E1 16728.532,E2 16728.532} C_VEL
LIN {X 0,Y 399.665,Z 504.052,A -85,B 0,C 180,E1 16726.546,E2 16726.546} C_VEL
LIN {X 0,Y 402.579,Z 508.289,A -85,B 0,C 180,E1 16724.366,E2 16724.366} C_VEL
LIN {X 0,Y 404.483,Z 510.087,A -85,B 0,C 180,E1 16723.188,E2 16723.188} C_VEL
LIN {X 0,Y 407.946,Z 514.615,A -85,B 0,C 180,E1 16721.197,E2 16721.197} C_VEL
LIN {X 0,Y 409.382,Z 516.372,A -85,B 0,C 180,E1 16720.451,E2 16720.451} C_VEL
LIN {X 0,Y 413.796,Z 522.081,A -85,B 0,C 180,E1 16718.34,E2 16718.34} C_VEL
LIN {X 0,Y 418.272,Z 527.966,A -85,B 0,C 180,E1 16716.433,E2 16716.433} C_VEL
LIN {X 0,Y 422.694,Z 533.91,A -85,B 0,C 180,E1 16714.724,E2 16714.724} C_VEL
LIN {X 0,Y 429.288,Z 542.973,A -85,B 0,C 180,E1 16712.424,E2 16712.424} C_VEL
LIN {X 0,Y 437.736,Z 555.27,A -85,B 0,C 180,E1 16709.794,E2 16709.794} C_VEL
LIN {X 0,Y 447.537,Z 570.474,A -85,B 0,C 180,E1 16707.08,E2 16707.08} C_VEL
LIN {X 0,Y 452.62,Z 579.187,A -85,B 0,C 180,E1 16705.771,E2 16705.771} C_VEL
LIN {X 0,Y 437.778,Z 811.734,A -85,B 0,C 180,E1 16701.991,E2 16701.991} C_VEL
LIN {X 0,Y 435.22,Z 836.444,A -85,B 0,C 180,E1 16701.45,E2 16701.45} C_VEL
LIN {X 0,Y 431.785,Z 859.352,A -85,B 0,C 180,E1 16700.757,E2 16700.757} C_VEL
LIN {X 0,Y 427.713,Z 881.467,A -85,B 0,C 180,E1 16699.91,E2 16699.91} C_VEL
LIN {X 0,Y 422.553,Z 904.253,A -85,B 0,C 180,E1 16698.807,E2 16698.807} C_VEL
LIN {X 0,Y 417.386,Z 924.079,A -85,B 0,C 180,E1 16697.65,E2 16697.65} C_VEL
LIN {X 0,Y 410.668,Z 946.697,A -85,B 0,C 180,E1 16696.059,E2 16696.059} C_VEL
LIN {X 0,Y 404.527,Z 965.271,A -85,B 0,C 180,E1 16694.494,E2 16694.494} C_VEL
LIN {X 0,Y 397.096,Z 985.913,A -85,B 0,C 180,E1 16692.441,E2 16692.441} C_VEL
LIN {X 0,Y 390.337,Z 1003.181,A -85,B 0,C 180,E1 16690.398,E2 16690.398} C_VEL
LIN {X 0,Y 383.237,Z 1020.542,A -85,B 0,C 180,E1 16688.006,E2 16688.006} C_VEL
LIN {X 0,Y 376.073,Z 1037.006,A -85,B 0,C 180,E1 16685.289,E2 16685.289} C_VEL
LIN {X 0,Y 369.528,Z 1051.999,A -85,B 0,C 180,E1 16682.396,E2 16682.396} C_VEL
LIN {X 0,Y 363.551,Z 1065.333,A -85,B 0,C 180,E1 16679.312,E2 16679.312} C_VEL
LIN {X 0,Y 358.474,Z 1077.021,A -85,B 0,C 180,E1 16676.149,E2 16676.149} C_VEL
LIN {X 0,Y 353.637,Z 1088.544,A -85,B 0,C 180,E1 16672.395,E2 16672.395} C_VEL
LIN {X 0,Y 350.296,Z 1097.224,A -85,B 0,C 180,E1 16668.99,E2 16668.99} C_VEL
LIN {X 0,Y 347.368,Z 1105.802,A -85,B 0,C 180,E1 16664.844,E2 16664.844} C_VEL
LIN {X 0,Y 345.746,Z 1111.522,A -85,B 0,C 180,E1 16661.341,E2 16661.341} C_VEL
LIN {X 0,Y 344.71,Z 1116.424,A -85,B 0,C 180,E1 16657.5,E2 16657.5} C_VEL
LIN {X 0,Y 344.207,Z 1119.695,A -85,B 0,C 180,E1 16653.664,E2 16653.664} C_VEL
LIN {X 0,Y 344.079,Z 1121.395,A -85,B 0,C 180,E1 16650.5,E2 16650.5} C_VEL
LIN {X 0,Y 344.032,Z 1122.206,A -85,B 0,C 180,E1 16647.001,E2 16647.001} C_VEL
LIN {X 0,Y 344.088,Z 1121.725,A -85,B 0,C 180,E1 16643.157,E2 16643.157} C_VEL
LIN {X 0,Y 344.282,Z 1120.13,A -85,B 0,C 180,E1 16639.795,E2 16639.795} C_VEL
LIN {X 0,Y 344.776,Z 1117.481,A -85,B 0,C 180,E1 16636.414,E2 16636.414} C_VEL
LIN {X 0,Y 345.978,Z 1112.872,A -85,B 0,C 180,E1 16632.335,E2 16632.335} C_VEL
LIN {X 0,Y 347.871,Z 1107.041,A -85,B 0,C 180,E1 16628.59,E2 16628.59} C_VEL
LIN {X 0,Y 350.847,Z 1099.474,A -85,B 0,C 180,E1 16624.691,E2 16624.691} C_VEL
LIN {X 0,Y 354.93,Z 1089.971,A -85,B 0,C 180,E1 16620.832,E2 16620.832} C_VEL
LIN {X 0,Y 359.728,Z 1079.737,A -85,B 0,C 180,E1 16617.368,E2 16617.368} C_VEL
LIN {X 0,Y 365.556,Z 1067.612,A -85,B 0,C 180,E1 16613.979,E2 16613.979} C_VEL
LIN {X 0,Y 371.392,Z 1055.677,A -85,B 0,C 180,E1 16611.148,E2 16611.148} C_VEL
LIN {X 0,Y 379.154,Z 1039.638,A -85,B 0,C 180,E1 16607.945,E2 16607.945} C_VEL
LIN {X 0,Y 385.761,Z 1025.606,A -85,B 0,C 180,E1 16605.586,E2 16605.586} C_VEL
LIN {X 0,Y 387.885,Z 1021.15,A -85,B 0,C 180,E1 16604.892,E2 16604.892} C_VEL
LIN {X 0,Y 389.491,Z 1016.18,A -85,B 0,C 180,E1 16604.044,E2 16604.044} C_VEL
LIN {X 0,Y 390.901,Z 1002.998,A -85,B 0,C 180,E1 16601.607,E2 16601.607} C_VEL
LIN {X 0,Y 392.473,Z 998.368,A -85,B 0,C 180,E1 16600.948,E2 16600.948} C_VEL
LIN {X 0,Y 400.535,Z 979.118,A -85,B 0,C 180,E1 16598.842,E2 16598.842} C_VEL
LIN {X 0,Y 407.652,Z 960.778,A -85,B 0,C 180,E1 16597.14,E2 16597.14} C_VEL
LIN {X 0,Y 415.368,Z 938.674,A -85,B 0,C 180,E1 16595.427,E2 16595.427} C_VEL
LIN {X 0,Y 421.304,Z 919.618,A -85,B 0,C 180,E1 16594.197,E2 16594.197} C_VEL
LIN {X 0,Y 427.699,Z 896.095,A -85,B 0,C 180,E1 16592.935,E2 16592.935} C_VEL
LIN {X 0,Y 432.673,Z 874.174,A -85,B 0,C 180,E1 16591.991,E2 16591.991} C_VEL
LIN {X 0,Y 437.206,Z 850.005,A -85,B 0,C 180,E1 16591.168,E2 16591.168} C_VEL
LIN {X 0,Y 440.422,Z 826.949,A -85,B 0,C 180,E1 16590.58,E2 16590.58} C_VEL
LIN {X 0,Y 442.822,Z 801.954,A -85,B 0,C 180,E1 16590.105,E2 16590.105} C_VEL
LIN {X 0,Y 457.594,Z 589.355,A -85,B 0,C 180,E1 16586.7,E2 16586.7} C_VEL
LIN {X 0,Y 449.769,Z 576.773,A -85,B 0,C 180,E1 16584.32,E2 16584.32} C_VEL
LIN {X 0,Y 443.039,Z 566.427,A -85,B 0,C 180,E1 16582.037,E2 16582.037} C_VEL
LIN {X 0,Y 435.565,Z 555.771,A -85,B 0,C 180,E1 16579.164,E2 16579.164} C_VEL
LIN {X 0,Y 431.791,Z 550.569,A -85,B 0,C 180,E1 16577.52,E2 16577.52} C_VEL
LIN {X 0,Y 429.103,Z 546.835,A -85,B 0,C 180,E1 16576.238,E2 16576.238} C_VEL
LIN {X 0,Y 425.643,Z 542.137,A -85,B 0,C 180,E1 16574.419,E2 16574.419} C_VEL
LIN {X 0,Y 422.162,Z 537.318,A -85,B 0,C 180,E1 16572.308,E2 16572.308} C_VEL
LIN {X 0,Y 419.038,Z 533.545,A -85,B 0,C 180,E1 16570.101,E2 16570.101} C_VEL
LIN {X 0,Y 418.013,Z 531.786,A -85,B 0,C 180,E1 16569.222,E2 16569.222} C_VEL
LIN {X 0,Y 415.187,Z 528.826,A -85,B 0,C 180,E1 16566.499,E2 16566.499} C_VEL
LIN {X 0,Y 413.865,Z 526.017,A -85,B 0,C 180,E1 16564.573,E2 16564.573} C_VEL
LIN {X 0,Y 411.859,Z 524.824,A -85,B 0,C 180,E1 16558.47,E2 16558.47} C_VEL
LIN {X 0,Y 414.033,Z 526.151,A -85,B 0,C 180,E1 16552.646,E2 16552.646} C_VEL
LIN {X 0,Y 416.019,Z 529.997,A -85,B 0,C 180,E1 16550.035,E2 16550.035} C_VEL
LIN {X 0,Y 418.463,Z 532.385,A -85,B 0,C 180,E1 16547.862,E2 16547.862} C_VEL
LIN {X 0,Y 421.501,Z 536.686,A -85,B 0,C 180,E1 16545.577,E2 16545.577} C_VEL
LIN {X 0,Y 422.841,Z 538.303,A -85,B 0,C 180,E1 16544.712,E2 16544.712} C_VEL
LIN {X 0,Y 427.054,Z 543.99,A -85,B 0,C 180,E1 16542.279,E2 16542.279} C_VEL
LIN {X 0,Y 431.903,Z 551.415,A -85,B 0,C 180,E1 16539.857,E2 16539.857} C_VEL
LIN {X 0,Y 437.758,Z 560.66,A -85,B 0,C 180,E1 16537.332,E2 16537.332} C_VEL
LIN {X 0,Y 445.743,Z 574.15,A -85,B 0,C 180,E1 16534.346,E2 16534.346} C_VEL
LIN {X 0,Y 453.461,Z 588.111,A -85,B 0,C 180,E1 16531.808,E2 16531.808} C_VEL
LIN {X 0,Y 457.368,Z 595.792,A -85,B 0,C 180,E1 16530.614,E2 16530.614} C_VEL
LIN {X 0,Y 442.267,Z 814.411,A -85,B 0,C 180,E1 16527.096,E2 16527.096} C_VEL
LIN {X 0,Y 439.723,Z 842.418,A -85,B 0,C 180,E1 16526.584,E2 16526.584} C_VEL
LIN {X 0,Y 436.504,Z 864.769,A -85,B 0,C 180,E1 16526.06,E2 16526.06} C_VEL
LIN {X 0,Y 431.594,Z 890.264,A -85,B 0,C 180,E1 16525.266,E2 16525.266} C_VEL
LIN {X 0,Y 426.609,Z 911.428,A -85,B 0,C 180,E1 16524.42,E2 16524.42} C_VEL
LIN {X 0,Y 419.751,Z 936.251,A -85,B 0,C 180,E1 16523.167,E2 16523.167} C_VEL
LIN {X 0,Y 413.402,Z 956.32,A -85,B 0,C 180,E1 16521.919,E2 16521.919} C_VEL
LIN {X 0,Y 405.337,Z 979.073,A -85,B 0,C 180,E1 16520.212,E2 16520.212} C_VEL
LIN {X 0,Y 398.197,Z 997.399,A -85,B 0,C 180,E1 16518.551,E2 16518.551} C_VEL
LIN {X 0,Y 389.895,Z 1017.272,A -85,B 0,C 180,E1 16516.425,E2 16516.425} C_VEL
LIN {X 0,Y 382.057,Z 1034.711,A -85,B 0,C 180,E1 16514.185,E2 16514.185} C_VEL
LIN {X 0,Y 373.942,Z 1052.222,A -85,B 0,C 180,E1 16511.539,E2 16511.539} C_VEL
LIN {X 0,Y 366.305,Z 1067.955,A -85,B 0,C 180,E1 16508.676,E2 16508.676} C_VEL
LIN {X 0,Y 359.286,Z 1082.518,A -85,B 0,C 180,E1 16505.567,E2 16505.567} C_VEL
LIN {X 0,Y 352.729,Z 1096.112,A -85,B 0,C 180,E1 16502.05,E2 16502.05} C_VEL
LIN {X 0,Y 347.277,Z 1108.137,A -85,B 0,C 180,E1 16498.364,E2 16498.364} C_VEL
LIN {X 0,Y 342.879,Z 1118.475,A -85,B 0,C 180,E1 16494.462,E2 16494.462} C_VEL
LIN {X 0,Y 339.829,Z 1126.853,A -85,B 0,C 180,E1 16490.664,E2 16490.664} C_VEL
LIN {X 0,Y 337.65,Z 1134.066,A -85,B 0,C 180,E1 16486.516,E2 16486.516} C_VEL
LIN {X 0,Y 336.567,Z 1139.027,A -85,B 0,C 180,E1 16482.874,E2 16482.874} C_VEL
LIN {X 0,Y 336.062,Z 1143.16,A -85,B 0,C 180,E1 16478.728,E2 16478.728} C_VEL
LIN {X 0,Y 335.976,Z 1145.344,A -85,B 0,C 180,E1 16475.122,E2 16475.122} C_VEL
LIN {X 0,Y 336.031,Z 1146.289,A -85,B 0,C 180,E1 16471.876,E2 16471.876} C_VEL
LIN {X 0,Y 336.04,Z 1146.227,A -85,B 0,C 180,E1 16468.636,E2 16468.636} C_VEL
LIN {X 0,Y 335.988,Z 1144.939,A -85,B 0,C 180,E1 16464.878,E2 16464.878} C_VEL
LIN {X 0,Y 336.079,Z 1141.944,A -85,B 0,C 180,E1 16460.927,E2 16460.927} C_VEL
LIN {X 0,Y 336.482,Z 1138.158,A -85,B 0,C 180,E1 16457.471,E2 16457.471} C_VEL
LIN {X 0,Y 337.593,Z 1132.389,A -85,B 0,C 180,E1 16453.481,E2 16453.481} C_VEL
LIN {X 0,Y 339.589,Z 1124.798,A -85,B 0,C 180,E1 16449.489,E2 16449.489} C_VEL
LIN {X 0,Y 342.659,Z 1115.622,A -85,B 0,C 180,E1 16445.521,E2 16445.521} C_VEL
LIN {X 0,Y 346.708,Z 1104.877,A -85,B 0,C 180,E1 16441.773,E2 16441.773} C_VEL
LIN {X 0,Y 351.669,Z 1093.005,A -85,B 0,C 180,E1 16438.264,E2 16438.264} C_VEL
LIN {X 0,Y 357.691,Z 1079.041,A -85,B 0,C 180,E1 16434.84,E2 16434.84} C_VEL
LIN {X 0,Y 363.729,Z 1065.417,A -85,B 0,C 180,E1 16431.991,E2 16431.991} C_VEL
LIN {X 0,Y 370.956,Z 1048.952,A -85,B 0,C 180,E1 16429.081,E2 16429.081} C_VEL
LIN {X 0,Y 377.705,Z 1033.189,A -85,B 0,C 180,E1 16426.713,E2 16426.713} C_VEL
LIN {X 0,Y 385.527,Z 1014.2,A -85,B 0,C 180,E1 16424.289,E2 16424.289} C_VEL
LIN {X 0,Y 392.708,Z 995.564,A -85,B 0,C 180,E1 16422.298,E2 16422.298} C_VEL
LIN {X 0,Y 400.162,Z 974.883,A -85,B 0,C 180,E1 16420.424,E2 16420.424} C_VEL
LIN {X 0,Y 406.765,Z 954.6,A -85,B 0,C 180,E1 16418.908,E2 16418.908} C_VEL
LIN {X 0,Y 413.385,Z 932.153,A -85,B 0,C 180,E1 16417.499,E2 16417.499} C_VEL
LIN {X 0,Y 419.199,Z 909.025,A -85,B 0,C 180,E1 16416.34,E2 16416.34} C_VEL
LIN {X 0,Y 424.426,Z 885.067,A -85,B 0,C 180,E1 16415.378,E2 16415.378} C_VEL
LIN {X 0,Y 428.522,Z 861.085,A -85,B 0,C 180,E1 16414.653,E2 16414.653} C_VEL
LIN {X 0,Y 431.706,Z 836.421,A -85,B 0,C 180,E1 16414.079,E2 16414.079} C_VEL
LIN {X 0,Y 435.15,Z 786.3,A -85,B 0,C 180,E1 16413.23,E2 16413.23} C_VEL
LIN {X 0,Y 447.82,Z 589.455,A -85,B 0,C 180,E1 16410.021,E2 16410.021} C_VEL
LIN {X 0,Y 438.452,Z 571.733,A -85,B 0,C 180,E1 16407.393,E2 16407.393} C_VEL
LIN {X 0,Y 430.622,Z 558.103,A -85,B 0,C 180,E1 16404.962,E2 16404.962} C_VEL
LIN {X 0,Y 423.828,Z 546.851,A -85,B 0,C 180,E1 16402.616,E2 16402.616} C_VEL
LIN {X 0,Y 416.956,Z 536.118,A -85,B 0,C 180,E1 16399.946,E2 16399.946} C_VEL
LIN {X 0,Y 413.624,Z 531.719,A -85,B 0,C 180,E1 16398.535,E2 16398.535} C_VEL
LIN {X 0,Y 410.45,Z 527.456,A -85,B 0,C 180,E1 16397.071,E2 16397.071} C_VEL
LIN {X 0,Y 406.607,Z 522.448,A -85,B 0,C 180,E1 16395.11,E2 16395.11} C_VEL
LIN {X 0,Y 403.177,Z 518.039,A -85,B 0,C 180,E1 16393.116,E2 16393.116} C_VEL
LIN {X 0,Y 402.193,Z 516.834,A -85,B 0,C 180,E1 16392.491,E2 16392.491} C_VEL
LIN {X 0,Y 399.02,Z 513.059,A -85,B 0,C 180,E1 16390.248,E2 16390.248} C_VEL
LIN {X 0,Y 398.025,Z 511.347,A -85,B 0,C 180,E1 16389.398,E2 16389.398} C_VEL
LIN {X 0,Y 394.874,Z 508.358,A -85,B 0,C 180,E1 16386.397,E2 16386.397} C_VEL
LIN {X 0,Y 393.396,Z 505.358,A -85,B 0,C 180,E1 16384.227,E2 16384.227} C_VEL
LIN {X 0,Y 391.391,Z 504.26,A -85,B 0,C 180,E1 16377.95,E2 16377.95} C_VEL
LIN {X 0,Y 393.575,Z 505.494,A -85,B 0,C 180,E1 16371.968,E2 16371.968} C_VEL
LIN {X 0,Y 395.482,Z 509.259,A -85,B 0,C 180,E1 16369.364,E2 16369.364} C_VEL
LIN {X 0,Y 398.341,Z 511.778,A -85,B 0,C 180,E1 16366.796,E2 16366.796} C_VEL
LIN {X 0,Y 401.298,Z 516.096,A -85,B 0,C 180,E1 16364.538,E2 16364.538} C_VEL
LIN {X 0,Y 403.056,Z 517.841,A -85,B 0,C 180,E1 16363.424,E2 16363.424} C_VEL
LIN {X 0,Y 406.6,Z 522.433,A -85,B 0,C 180,E1 16361.356,E2 16361.356} C_VEL
LIN {X 0,Y 411.944,Z 529.459,A -85,B 0,C 180,E1 16358.686,E2 16358.686} C_VEL
LIN {X 0,Y 416.573,Z 535.684,A -85,B 0,C 180,E1 16356.669,E2 16356.669} C_VEL
LIN {X 0,Y 422.478,Z 543.641,A -85,B 0,C 180,E1 16354.386,E2 16354.386} C_VEL
LIN {X 0,Y 430.778,Z 555.64,A -85,B 0,C 180,E1 16351.549,E2 16351.549} C_VEL
LIN {X 0,Y 439.743,Z 569.335,A -85,B 0,C 180,E1 16348.849,E2 16348.849} C_VEL
LIN {X 0,Y 448.127,Z 583.006,A -85,B 0,C 180,E1 16346.576,E2 16346.576} C_VEL
LIN {X 0,Y 433.054,Z 812.436,A -85,B 0,C 180,E1 16342.836,E2 16342.836} C_VEL
LIN {X 0,Y 430.361,Z 837.434,A -85,B 0,C 180,E1 16342.283,E2 16342.283} C_VEL
LIN {X 0,Y 426.902,Z 859.903,A -85,B 0,C 180,E1 16341.6,E2 16341.6} C_VEL
LIN {X 0,Y 422.643,Z 882.434,A -85,B 0,C 180,E1 16340.734,E2 16340.734} C_VEL
LIN {X 0,Y 417.351,Z 905.061,A -85,B 0,C 180,E1 16339.629,E2 16339.629} C_VEL
LIN {X 0,Y 412.055,Z 924.83,A -85,B 0,C 180,E1 16338.47,E2 16338.47} C_VEL
LIN {X 0,Y 405.152,Z 947.372,A -85,B 0,C 180,E1 16336.873,E2 16336.873} C_VEL
LIN {X 0,Y 398.818,Z 965.984,A -85,B 0,C 180,E1 16335.294,E2 16335.294} C_VEL
LIN {X 0,Y 390.96,Z 987.084,A -85,B 0,C 180,E1 16333.168,E2 16333.168} C_VEL
LIN {X 0,Y 384.238,Z 1003.731,A -85,B 0,C 180,E1 16331.176,E2 16331.176} C_VEL
LIN {X 0,Y 376.791,Z 1021.304,A -85,B 0,C 180,E1 16328.722,E2 16328.722} C_VEL
LIN {X 0,Y 369.769,Z 1036.899,A -85,B 0,C 180,E1 16326.121,E2 16326.121} C_VEL
LIN {X 0,Y 363.032,Z 1051.72,A -85,B 0,C 180,E1 16323.237,E2 16323.237} C_VEL
LIN {X 0,Y 356.5,Z 1065.774,A -85,B 0,C 180,E1 16319.95,E2 16319.95} C_VEL
LIN {X 0,Y 351.207,Z 1077.448,A -85,B 0,C 180,E1 16316.733,E2 16316.733} C_VEL
LIN {X 0,Y 346.204,Z 1088.828,A -85,B 0,C 180,E1 16312.948,E2 16312.948} C_VEL
LIN {X 0,Y 342.65,Z 1097.61,A -85,B 0,C 180,E1 16309.431,E2 16309.431} C_VEL
LIN {X 0,Y 339.567,Z 1106.163,A -85,B 0,C 180,E1 16305.193,E2 16305.193} C_VEL
LIN {X 0,Y 337.918,Z 1111.623,A -85,B 0,C 180,E1 16301.781,E2 16301.781} C_VEL
LIN {X 0,Y 336.784,Z 1116.568,A -85,B 0,C 180,E1 16297.85,E2 16297.85} C_VEL
LIN {X 0,Y 336.234,Z 1119.897,A -85,B 0,C 180,E1 16293.922,E2 16293.922} C_VEL
LIN {X 0,Y 336.08,Z 1121.63,A -85,B 0,C 180,E1 16290.682,E2 16290.682} C_VEL
LIN {X 0,Y 336.037,Z 1122.45,A -85,B 0,C 180,E1 16287.271,E2 16287.271} C_VEL
LIN {X 0,Y 336.099,Z 1122.126,A -85,B 0,C 180,E1 16283.337,E2 16283.337} C_VEL
LIN {X 0,Y 336.318,Z 1120.39,A -85,B 0,C 180,E1 16279.551,E2 16279.551} C_VEL
LIN {X 0,Y 336.854,Z 1117.728,A -85,B 0,C 180,E1 16276.083,E2 16276.083} C_VEL
LIN {X 0,Y 338.16,Z 1113.101,A -85,B 0,C 180,E1 16271.912,E2 16271.912} C_VEL
LIN {X 0,Y 340.196,Z 1107.259,A -85,B 0,C 180,E1 16268.082,E2 16268.082} C_VEL
LIN {X 0,Y 343.37,Z 1099.682,A -85,B 0,C 180,E1 16264.1,E2 16264.1} C_VEL
LIN {X 0,Y 347.694,Z 1090.154,A -85,B 0,C 180,E1 16260.165,E2 16260.165} C_VEL
LIN {X 0,Y 352.744,Z 1079.906,A -85,B 0,C 180,E1 16256.639,E2 16256.639} C_VEL
LIN {X 0,Y 358.854,Z 1067.752,A -85,B 0,C 180,E1 16253.197,E2 16253.197} C_VEL
LIN {X 0,Y 364.946,Z 1055.802,A -85,B 0,C 180,E1 16250.329,E2 16250.329} C_VEL
LIN {X 0,Y 373.036,Z 1039.728,A -85,B 0,C 180,E1 16247.092,E2 16247.092} C_VEL
LIN {X 0,Y 379.892,Z 1025.675,A -85,B 0,C 180,E1 16244.712,E2 16244.712} C_VEL
LIN {X 0,Y 388.056,Z 1008.32,A -85,B 0,C 180,E1 16242.201,E2 16242.201} C_VEL
LIN {X 0,Y 392.473,Z 998.368,A -85,B 0,C 180,E1 16240.948,E2 16240.948} C_VEL
LIN {X 0,Y 394.243,Z 992.907,A -85,B 0,C 180,E1 16240.186,E2 16240.186} C_VEL
LIN {X 0,Y 395.996,Z 979.295,A -85,B 0,C 180,E1 16238.053,E2 16238.053} C_VEL
LIN {X 0,Y 397.784,Z 973.469,A -85,B 0,C 180,E1 16237.361,E2 16237.361} C_VEL
LIN {X 0,Y 405.871,Z 952.289,A -85,B 0,C 180,E1 16235.522,E2 16235.522} C_VEL
LIN {X 0,Y 412.203,Z 934.02,A -85,B 0,C 180,E1 16234.19,E2 16234.19} C_VEL
LIN {X 0,Y 419.412,Z 910.468,A -85,B 0,C 180,E1 16232.764,E2 16232.764} C_VEL
LIN {X 0,Y 424.606,Z 890.613,A -85,B 0,C 180,E1 16231.776,E2 16231.776} C_VEL
LIN {X 0,Y 429.852,Z 867.163,A -85,B 0,C 180,E1 16230.824,E2 16230.824} C_VEL
LIN {X 0,Y 433.882,Z 843.98,A -85,B 0,C 180,E1 16230.102,E2 16230.102} C_VEL
LIN {X 0,Y 437.16,Z 819.503,A -85,B 0,C 180,E1 16229.523,E2 16229.523} C_VEL
LIN {X 0,Y 440.936,Z 769.665,A -85,B 0,C 180,E1 16228.69,E2 16228.69} C_VEL
LIN {X 0,Y 453.512,Z 593.741,A -85,B 0,C 180,E1 16225.866,E2 16225.866} C_VEL
LIN {X 0,Y 444.439,Z 579.043,A -85,B 0,C 180,E1 16222.941,E2 16222.941} C_VEL
LIN {X 0,Y 437.421,Z 568.561,A -85,B 0,C 180,E1 16220.367,E2 16220.367} C_VEL
LIN {X 0,Y 431.367,Z 559.755,A -85,B 0,C 180,E1 16217.817,E2 16217.817} C_VEL
LIN {X 0,Y 427.206,Z 554.055,A -85,B 0,C 180,E1 16215.823,E2 16215.823} C_VEL
LIN {X 0,Y 424.071,Z 549.691,A -85,B 0,C 180,E1 16214.125,E2 16214.125} C_VEL
LIN {X 0,Y 420.561,Z 544.843,A -85,B 0,C 180,E1 16211.938,E2 16211.938} C_VEL
LIN {X 0,Y 417.482,Z 540.792,A -85,B 0,C 180,E1 16209.651,E2 16209.651} C_VEL
LIN {X 0,Y 416.709,Z 539.555,A -85,B 0,C 180,E1 16208.973,E2 16208.973} C_VEL
LIN {X 0,Y 413.874,Z 536.331,A -85,B 0,C 180,E1 16206.102,E2 16206.102} C_VEL
LIN {X 0,Y 412.795,Z 533.925,A -85,B 0,C 180,E1 16204.446,E2 16204.446} C_VEL
LIN {X 0,Y 410.883,Z 532.764,A -85,B 0,C 180,E1 16198.466,E2 16198.466} C_VEL
LIN {X 0,Y 412.96,Z 534.098,A -85,B 0,C 180,E1 16192.767,E2 16192.767} C_VEL
LIN {X 0,Y 415.047,Z 538.038,A -85,B 0,C 180,E1 16190.011,E2 16190.011} C_VEL
LIN {X 0,Y 417.237,Z 540.245,A -85,B 0,C 180,E1 16188.036,E2 16188.036} C_VEL
LIN {X 0,Y 420.333,Z 544.587,A -85,B 0,C 180,E1 16185.676,E2 16185.676} C_VEL
LIN {X 0,Y 421.542,Z 546.201,A -85,B 0,C 180,E1 16184.875,E2 16184.875} C_VEL
LIN {X 0,Y 425.582,Z 551.732,A -85,B 0,C 180,E1 16182.498,E2 16182.498} C_VEL
LIN {X 0,Y 430.151,Z 558.91,A -85,B 0,C 180,E1 16180.161,E2 16180.161} C_VEL
LIN {X 0,Y 435.985,Z 568.316,A -85,B 0,C 180,E1 16177.587,E2 16177.587} C_VEL
LIN {X 0,Y 443.839,Z 581.997,A -85,B 0,C 180,E1 16174.585,E2 16174.585} C_VEL
LIN {X 0,Y 450.991,Z 595.245,A -85,B 0,C 180,E1 16172.18,E2 16172.18} C_VEL
LIN {X 0,Y 453.324,Z 599.901,A -85,B 0,C 180,E1 16171.442,E2 16171.442} C_VEL
LIN {X 0,Y 437.721,Z 819.803,A -85,B 0,C 180,E1 16167.9,E2 16167.9} C_VEL
LIN {X 0,Y 435.233,Z 844.322,A -85,B 0,C 180,E1 16167.435,E2 16167.435} C_VEL
LIN {X 0,Y 431.517,Z 868.882,A -85,B 0,C 180,E1 16166.842,E2 16166.842} C_VEL
LIN {X 0,Y 426.784,Z 891.876,A -85,B 0,C 180,E1 16166.1,E2 16166.1} C_VEL
LIN {X 0,Y 421.668,Z 912.917,A -85,B 0,C 180,E1 16165.25,E2 16165.25} C_VEL
LIN {X 0,Y 414.967,Z 936.352,A -85,B 0,C 180,E1 16164.059,E2 16164.059} C_VEL
LIN {X 0,Y 408.47,Z 956.364,A -85,B 0,C 180,E1 16162.813,E2 16162.813} C_VEL
LIN {X 0,Y 399.896,Z 979.801,A -85,B 0,C 180,E1 16161.043,E2 16161.043} C_VEL
LIN {X 0,Y 392.573,Z 998.033,A -85,B 0,C 180,E1 16159.377,E2 16159.377} C_VEL
LIN {X 0,Y 383.519,Z 1018.864,A -85,B 0,C 180,E1 16157.106,E2 16157.106} C_VEL
LIN {X 0,Y 375.882,Z 1035.304,A -85,B 0,C 180,E1 16154.96,E2 16154.96} C_VEL
LIN {X 0,Y 367.359,Z 1052.964,A -85,B 0,C 180,E1 16152.239,E2 16152.239} C_VEL
LIN {X 0,Y 359.913,Z 1067.757,A -85,B 0,C 180,E1 16149.509,E2 16149.509} C_VEL
LIN {X 0,Y 352.582,Z 1082.356,A -85,B 0,C 180,E1 16146.349,E2 16146.349} C_VEL
LIN {X 0,Y 345.956,Z 1095.46,A -85,B 0,C 180,E1 16142.913,E2 16142.913} C_VEL
LIN {X 0,Y 340.47,Z 1106.898,A -85,B 0,C 180,E1 16139.37,E2 16139.37} C_VEL
LIN {X 0,Y 335.727,Z 1117.43,A -85,B 0,C 180,E1 16135.396,E2 16135.396} C_VEL
LIN {X 0,Y 332.494,Z 1125.569,A -85,B 0,C 180,E1 16131.683,E2 16131.683} C_VEL
LIN {X 0,Y 329.875,Z 1133.559,A -85,B 0,C 180,E1 16127.099,E2 16127.099} C_VEL
LIN {X 0,Y 328.673,Z 1138.561,A -85,B 0,C 180,E1 16123.368,E2 16123.368} C_VEL
LIN {X 0,Y 328.075,Z 1142.802,A -85,B 0,C 180,E1 16119.077,E2 16119.077} C_VEL
LIN {X 0,Y 327.979,Z 1144.999,A -85,B 0,C 180,E1 16115.423,E2 16115.423} C_VEL
LIN {X 0,Y 328.029,Z 1145.984,A -85,B 0,C 180,E1 16112.096,E2 16112.096} C_VEL
LIN {X 0,Y 328.044,Z 1145.962,A -85,B 0,C 180,E1 16108.777,E2 16108.777} C_VEL
LIN {X 0,Y 327.997,Z 1144.787,A -85,B 0,C 180,E1 16105.103,E2 16105.103} C_VEL
LIN {X 0,Y 328.074,Z 1141.958,A -85,B 0,C 180,E1 16101.058,E2 16101.058} C_VEL
LIN {X 0,Y 328.468,Z 1138.258,A -85,B 0,C 180,E1 16097.518,E2 16097.518} C_VEL
LIN {X 0,Y 329.46,Z 1133.136,A -85,B 0,C 180,E1 16093.787,E2 16093.787} C_VEL
LIN {X 0,Y 331.53,Z 1125.53,A -85,B 0,C 180,E1 16089.521,E2 16089.521} C_VEL
LIN {X 0,Y 334.311,Z 1117.339,A -85,B 0,C 180,E1 16085.811,E2 16085.811} C_VEL
LIN {X 0,Y 338.816,Z 1105.913,A -85,B 0,C 180,E1 16081.575,E2 16081.575} C_VEL
LIN {X 0,Y 343.559,Z 1094.898,A -85,B 0,C 180,E1 16078.194,E2 16078.194} C_VEL
LIN {X 0,Y 350.048,Z 1080.539,A -85,B 0,C 180,E1 16074.497,E2 16074.497} C_VEL
LIN {X 0,Y 356.469,Z 1066.547,A -85,B 0,C 180,E1 16071.486,E2 16071.486} C_VEL
LIN {X 0,Y 364.306,Z 1049.423,A -85,B 0,C 180,E1 16068.378,E2 16068.378} C_VEL
LIN {X 0,Y 371.282,Z 1033.679,A -85,B 0,C 180,E1 16065.976,E2 16065.976} C_VEL
LIN {X 0,Y 379.311,Z 1014.907,A -85,B 0,C 180,E1 16063.538,E2 16063.538} C_VEL
LIN {X 0,Y 386.598,Z 996.594,A -85,B 0,C 180,E1 16061.554,E2 16061.554} C_VEL
LIN {X 0,Y 394.242,Z 976.148,A -85,B 0,C 180,E1 16059.668,E2 16059.668} C_VEL
LIN {X 0,Y 401.349,Z 954.978,A -85,B 0,C 180,E1 16058.07,E2 16058.07} C_VEL
LIN {X 0,Y 407.553,Z 934.553,A -85,B 0,C 180,E1 16056.772,E2 16056.772} C_VEL
LIN {X 0,Y 413.682,Z 911.372,A -85,B 0,C 180,E1 16055.576,E2 16055.576} C_VEL
LIN {X 0,Y 418.439,Z 890.515,A -85,B 0,C 180,E1 16054.713,E2 16054.713} C_VEL
LIN {X 0,Y 423.156,Z 865.33,A -85,B 0,C 180,E1 16053.897,E2 16053.897} C_VEL
LIN {X 0,Y 426.285,Z 842.955,A -85,B 0,C 180,E1 16053.35,E2 16053.35} C_VEL
LIN {X 0,Y 428.708,Z 815.708,A -85,B 0,C 180,E1 16052.836,E2 16052.836} C_VEL
LIN {X 0,Y 443.183,Z 596.885,A -85,B 0,C 180,E1 16049.264,E2 16049.264} C_VEL
LIN {X 0,Y 443.311,Z 593.153,A -85,B 0,C 180,E1 16049.176,E2 16049.176} C_VEL
LIN {X 0,Y 435.069,Z 577.417,A -85,B 0,C 180,E1 16046.773,E2 16046.773} C_VEL
LIN {X 0,Y 427.71,Z 564.327,A -85,B 0,C 180,E1 16044.406,E2 16044.406} C_VEL
LIN {X 0,Y 420.493,Z 552.13,A -85,B 0,C 180,E1 16041.811,E2 16041.811} C_VEL
LIN {X 0,Y 413.929,Z 541.919,A -85,B 0,C 180,E1 16039.143,E2 16039.143} C_VEL
LIN {X 0,Y 408.626,Z 534.837,A -85,B 0,C 180,E1 16036.709,E2 16036.709} C_VEL
LIN {X 0,Y 404.865,Z 529.887,A -85,B 0,C 180,E1 16034.737,E2 16034.737} C_VEL
LIN {X 0,Y 401.437,Z 525.201,A -85,B 0,C 180,E1 16032.661,E2 16032.661} C_VEL
LIN {X 0,Y 397.68,Z 520.745,A -85,B 0,C 180,E1 16029.991,E2 16029.991} C_VEL
LIN {X 0,Y 396.701,Z 519.118,A -85,B 0,C 180,E1 16029.137,E2 16029.137} C_VEL
LIN {X 0,Y 393.543,Z 515.866,A -85,B 0,C 180,E1 16025.979,E2 16025.979} C_VEL
LIN {X 0,Y 392.325,Z 513.252,A -85,B 0,C 180,E1 16024.092,E2 16024.092} C_VEL
LIN {X 0,Y 390.422,Z 512.201,A -85,B 0,C 180,E1 16017.798,E2 16017.798} C_VEL
LIN {X 0,Y 392.506,Z 513.394,A -85,B 0,C 180,E1 16012.093,E2 16012.093} C_VEL
LIN {X 0,Y 394.377,Z 517.145,A -85,B 0,C 180,E1 16009.482,E2 16009.482} C_VEL
LIN {X 0,Y 397.103,Z 519.667,A -85,B 0,C 180,E1 16006.976,E2 16006.976} C_VEL
LIN {X 0,Y 400.126,Z 524.004,A -85,B 0,C 180,E1 16004.64,E2 16004.64} C_VEL
LIN {X 0,Y 401.637,Z 525.588,A -85,B 0,C 180,E1 16003.661,E2 16003.661} C_VEL
LIN {X 0,Y 405.257,Z 530.25,A -85,B 0,C 180,E1 16001.515,E2 16001.515} C_VEL
LIN {X 0,Y 410.386,Z 537.263,A -85,B 0,C 180,E1 15998.9,E2 15998.9} C_VEL
LIN {X 0,Y 414.572,Z 542.951,A -85,B 0,C 180,E1 15997.038,E2 15997.038} C_VEL
LIN {X 0,Y 420.398,Z 550.991,A -85,B 0,C 180,E1 15994.727,E2 15994.727} C_VEL
LIN {X 0,Y 428.542,Z 562.943,A -85,B 0,C 180,E1 15991.88,E2 15991.88} C_VEL
LIN {X 0,Y 437.479,Z 576.961,A -85,B 0,C 180,E1 15989.128,E2 15989.128} C_VEL
LIN {X 0,Y 443.693,Z 587.297,A -85,B 0,C 180,E1 15987.389,E2 15987.389} C_VEL
LIN {X 0,Y 428.424,Z 813.121,A -85,B 0,C 180,E1 15983.699,E2 15983.699} C_VEL
LIN {X 0,Y 425.574,Z 838.544,A -85,B 0,C 180,E1 15983.131,E2 15983.131} C_VEL
LIN {X 0,Y 422.095,Z 860.554,A -85,B 0,C 180,E1 15982.458,E2 15982.458} C_VEL
LIN {X 0,Y 417.66,Z 883.38,A -85,B 0,C 180,E1 15981.578,E2 15981.578} C_VEL
LIN {X 0,Y 412.238,Z 905.868,A -85,B 0,C 180,E1 15980.472,E2 15980.472} C_VEL
LIN {X 0,Y 406.255,Z 927.558,A -85,B 0,C 180,E1 15979.186,E2 15979.186} C_VEL
LIN {X 0,Y 399.722,Z 948.043,A -85,B 0,C 180,E1 15977.709,E2 15977.709} C_VEL
LIN {X 0,Y 393.191,Z 966.691,A -85,B 0,C 180,E1 15976.117,E2 15976.117} C_VEL
LIN {X 0,Y 384.888,Z 988.251,A -85,B 0,C 180,E1 15973.919,E2 15973.919} C_VEL
LIN {X 0,Y 377.981,Z 1004.823,A -85,B 0,C 180,E1 15971.909,E2 15971.909} C_VEL
LIN {X 0,Y 369.783,Z 1023.373,A -85,B 0,C 180,E1 15969.252,E2 15969.252} C_VEL
LIN {X 0,Y 362.877,Z 1038.215,A -85,B 0,C 180,E1 15966.722,E2 15966.722} C_VEL
LIN {X 0,Y 355.596,Z 1053.616,A -85,B 0,C 180,E1 15963.638,E2 15963.638} C_VEL
LIN {X 0,Y 349.197,Z 1066.835,A -85,B 0,C 180,E1 15960.453,E2 15960.453} C_VEL
LIN {X 0,Y 343.484,Z 1078.993,A -85,B 0,C 180,E1 15957.008,E2 15957.008} C_VEL
LIN {X 0,Y 338.494,Z 1089.799,A -85,B 0,C 180,E1 15953.266,E2 15953.266} C_VEL
LIN {X 0,Y 334.568,Z 1099.178,A -85,B 0,C 180,E1 15949.374,E2 15949.374} C_VEL
LIN {X 0,Y 331.569,Z 1107.112,A -85,B 0,C 180,E1 15945.21,E2 15945.21} C_VEL
LIN {X 0,Y 329.834,Z 1112.712,A -85,B 0,C 180,E1 15941.542,E2 15941.542} C_VEL
LIN {X 0,Y 328.662,Z 1117.695,A -85,B 0,C 180,E1 15937.165,E2 15937.165} C_VEL
LIN {X 0,Y 328.222,Z 1120.43,A -85,B 0,C 180,E1 15933.668,E2 15933.668} C_VEL
LIN {X 0,Y 328.098,Z 1122.13,A -85,B 0,C 180,E1 15930.175,E2 15930.175} C_VEL
LIN {X 0,Y 328.047,Z 1122.803,A -85,B 0,C 180,E1 15925.98,E2 15925.98} C_VEL
LIN {X 0,Y 328.131,Z 1122.069,A -85,B 0,C 180,E1 15922.295,E2 15922.295} C_VEL
LIN {X 0,Y 328.424,Z 1120.322,A -85,B 0,C 180,E1 15918.764,E2 15918.764} C_VEL
LIN {X 0,Y 329.272,Z 1116.844,A -85,B 0,C 180,E1 15914.501,E2 15914.501} C_VEL
LIN {X 0,Y 330.868,Z 1111.84,A -85,B 0,C 180,E1 15910.4,E2 15910.4} C_VEL
LIN {X 0,Y 333.46,Z 1105.402,A -85,B 0,C 180,E1 15906.309,E2 15906.309} C_VEL
LIN {X 0,Y 337.171,Z 1097.116,A -85,B 0,C 180,E1 15902.252,E2 15902.252} C_VEL
LIN {X 0,Y 341.655,Z 1088.072,A -85,B 0,C 180,E1 15898.605,E2 15898.605} C_VEL
LIN {X 0,Y 347.744,Z 1076.328,A -85,B 0,C 180,E1 15894.747,E2 15894.747} C_VEL
LIN {X 0,Y 353.912,Z 1064.743,A -85,B 0,C 180,E1 15891.57,E2 15891.57} C_VEL
LIN {X 0,Y 361.673,Z 1050.079,A -85,B 0,C 180,E1 15888.22,E2 15888.22} C_VEL
LIN {X 0,Y 368.728,Z 1036.448,A -85,B 0,C 180,E1 15885.603,E2 15885.603} C_VEL
LIN {X 0,Y 377.4,Z 1019.086,A -85,B 0,C 180,E1 15882.786,E2 15882.786} C_VEL
LIN {X 0,Y 384.952,Z 1003.038,A -85,B 0,C 180,E1 15880.607,E2 15880.607} C_VEL
LIN {X 0,Y 393.256,Z 984.438,A -85,B 0,C 180,E1 15878.453,E2 15878.453} C_VEL
LIN {X 0,Y 397.784,Z 973.469,A -85,B 0,C 180,E1 15877.361,E2 15877.361} C_VEL
LIN {X 0,Y 399.581,Z 967.551,A -85,B 0,C 180,E1 15876.685,E2 15876.685} C_VEL
LIN {X 0,Y 401.689,Z 951.986,A -85,B 0,C 180,E1 15874.642,E2 15874.642} C_VEL
LIN {X 0,Y 403.244,Z 946.599,A -85,B 0,C 180,E1 15874.135,E2 15874.135} C_VEL
LIN {X 0,Y 410.787,Z 924.303,A -85,B 0,C 180,E1 15872.627,E2 15872.627} C_VEL
LIN {X 0,Y 416.941,Z 903.502,A -85,B 0,C 180,E1 15871.462,E2 15871.462} C_VEL
LIN {X 0,Y 423.071,Z 878.953,A -85,B 0,C 180,E1 15870.351,E2 15870.351} C_VEL
LIN {X 0,Y 427.385,Z 858.015,A -85,B 0,C 180,E1 15869.603,E2 15869.603} C_VEL
LIN {X 0,Y 431.412,Z 833.065,A -85,B 0,C 180,E1 15868.91,E2 15868.91} C_VEL
LIN {X 0,Y 433.904,Z 810.623,A -85,B 0,C 180,E1 15868.453,E2 15868.453} C_VEL
LIN {X 0,Y 449.579,Z 598.32,A -85,B 0,C 180,E1 15865.038,E2 15865.038} C_VEL
LIN {X 0,Y 441.086,Z 584.456,A -85,B 0,C 180,E1 15862.175,E2 15862.175} C_VEL
LIN {X 0,Y 434.083,Z 573.89,A -85,B 0,C 180,E1 15859.477,E2 15859.477} C_VEL
LIN {X 0,Y 428.835,Z 566.217,A -85,B 0,C 180,E1 15857.155,E2 15857.155} C_VEL
LIN {X 0,Y 425.582,Z 561.59,A -85,B 0,C 180,E1 15855.536,E2 15855.536} C_VEL
LIN {X 0,Y 422.512,Z 557.241,A -85,B 0,C 180,E1 15853.829,E2 15853.829} C_VEL
LIN {X 0,Y 419.18,Z 552.545,A -85,B 0,C 180,E1 15851.698,E2 15851.698} C_VEL
LIN {X 0,Y 416.099,Z 548.331,A -85,B 0,C 180,E1 15849.335,E2 15849.335} C_VEL
LIN {X 0,Y 415.414,Z 547.321,A -85,B 0,C 180,E1 15848.722,E2 15848.722} C_VEL
LIN {X 0,Y 412.68,Z 544.029,A -85,B 0,C 180,E1 15845.841,E2 15845.841} C_VEL
LIN {X 0,Y 411.728,Z 541.833,A -85,B 0,C 180,E1 15844.318,E2 15844.318} C_VEL
LIN {X 0,Y 409.908,Z 540.704,A -85,B 0,C 180,E1 15838.462,E2 15838.462} C_VEL
LIN {X 0,Y 411.888,Z 542.039,A -85,B 0,C 180,E1 15832.888,E2 15832.888} C_VEL
LIN {X 0,Y 414.075,Z 546.073,A -85,B 0,C 180,E1 15829.987,E2 15829.987} C_VEL
LIN {X 0,Y 415.942,Z 547.948,A -85,B 0,C 180,E1 15828.28,E2 15828.28} C_VEL
LIN {X 0,Y 418.966,Z 552.292,A -85,B 0,C 180,E1 15825.911,E2 15825.911} C_VEL
LIN {X 0,Y 420.248,Z 554.089,A -85,B 0,C 180,E1 15825.039,E2 15825.039} C_VEL
LIN {X 0,Y 424.001,Z 559.287,A -85,B 0,C 180,E1 15822.785,E2 15822.785} C_VEL
LIN {X 0,Y 428.413,Z 566.401,A -85,B 0,C 180,E1 15820.468,E2 15820.468} C_VEL
LIN {X 0,Y 434.141,Z 575.83,A -85,B 0,C 180,E1 15817.879,E2 15817.879} C_VEL
LIN {X 0,Y 441.609,Z 589.2,A -85,B 0,C 180,E1 15814.95,E2 15814.95} C_VEL
LIN {X 0,Y 448.451,Z 602.188,A -85,B 0,C 180,E1 15812.585,E2 15812.585} C_VEL
LIN {X 0,Y 449.357,Z 604.27,A -85,B 0,C 180,E1 15812.279,E2 15812.279} C_VEL
LIN {X 0,Y 433.26,Z 824.056,A -85,B 0,C 180,E1 15808.733,E2 15808.733} C_VEL
LIN {X 0,Y 430.829,Z 846.33,A -85,B 0,C 180,E1 15808.3,E2 15808.3} C_VEL
LIN {X 0,Y 426.521,Z 872.638,A -85,B 0,C 180,E1 15807.638,E2 15807.638} C_VEL
LIN {X 0,Y 422.184,Z 892.969,A -85,B 0,C 180,E1 15806.973,E2 15806.973} C_VEL
LIN {X 0,Y 416.377,Z 916.089,A -85,B 0,C 180,E1 15806.024,E2 15806.024} C_VEL
LIN {X 0,Y 409.647,Z 938.458,A -85,B 0,C 180,E1 15804.854,E2 15804.854} C_VEL
LIN {X 0,Y 402.433,Z 959.932,A -85,B 0,C 180,E1 15803.492,E2 15803.492} C_VEL
LIN {X 0,Y 394.246,Z 981.267,A -85,B 0,C 180,E1 15801.835,E2 15801.835} C_VEL
LIN {X 0,Y 386.193,Z 1000.675,A -85,B 0,C 180,E1 15800.03,E2 15800.03} C_VEL
LIN {X 0,Y 377.199,Z 1020.456,A -85,B 0,C 180,E1 15797.809,E2 15797.809} C_VEL
LIN {X 0,Y 369.096,Z 1037.321,A -85,B 0,C 180,E1 15795.56,E2 15795.56} C_VEL
LIN {X 0,Y 360.406,Z 1054.513,A -85,B 0,C 180,E1 15792.822,E2 15792.822} C_VEL
LIN {X 0,Y 353.167,Z 1068.388,A -85,B 0,C 180,E1 15790.205,E2 15790.205} C_VEL
LIN {X 0,Y 345.233,Z 1083.489,A -85,B 0,C 180,E1 15786.836,E2 15786.836} C_VEL
LIN {X 0,Y 338.722,Z 1095.855,A -85,B 0,C 180,E1 15783.506,E2 15783.506} C_VEL
LIN {X 0,Y 332.783,Z 1107.731,A -85,B 0,C 180,E1 15779.72,E2 15779.72} C_VEL
LIN {X 0,Y 327.897,Z 1118.038,A -85,B 0,C 180,E1 15775.659,E2 15775.659} C_VEL
LIN {X 0,Y 324.333,Z 1126.733,A -85,B 0,C 180,E1 15771.523,E2 15771.523} C_VEL
LIN {X 0,Y 321.883,Z 1133.837,A -85,B 0,C 180,E1 15767.164,E2 15767.164} C_VEL
LIN {X 0,Y 320.619,Z 1138.948,A -85,B 0,C 180,E1 15763.159,E2 15763.159} C_VEL
LIN {X 0,Y 320.065,Z 1142.864,A -85,B 0,C 180,E1 15758.805,E2 15758.805} C_VEL
LIN {X 0,Y 319.982,Z 1144.797,A -85,B 0,C 180,E1 15755.379,E2 15755.379} C_VEL
LIN {X 0,Y 320.033,Z 1145.703,A -85,B 0,C 180,E1 15752.149,E2 15752.149} C_VEL
LIN {X 0,Y 320.049,Z 1145.673,A -85,B 0,C 180,E1 15748.747,E2 15748.747} C_VEL
LIN {X 0,Y 319.997,Z 1144.489,A -85,B 0,C 180,E1 15744.981,E2 15744.981} C_VEL
LIN {X 0,Y 320.088,Z 1141.608,A -85,B 0,C 180,E1 15740.796,E2 15740.796} C_VEL
LIN {X 0,Y 320.526,Z 1137.93,A -85,B 0,C 180,E1 15737.204,E2 15737.204} C_VEL
LIN {X 0,Y 321.669,Z 1132.534,A -85,B 0,C 180,E1 15733.197,E2 15733.197} C_VEL
LIN {X 0,Y 323.933,Z 1124.807,A -85,B 0,C 180,E1 15728.829,E2 15728.829} C_VEL
LIN {X 0,Y 326.939,Z 1116.552,A -85,B 0,C 180,E1 15725.036,E2 15725.036} C_VEL
LIN {X 0,Y 331.69,Z 1105.148,A -85,B 0,C 180,E1 15720.767,E2 15720.767} C_VEL
LIN {X 0,Y 336.765,Z 1093.957,A -85,B 0,C 180,E1 15717.291,E2 15717.291} C_VEL
LIN {X 0,Y 343.537,Z 1079.613,A -85,B 0,C 180,E1 15713.576,E2 15713.576} C_VEL
LIN {X 0,Y 350.001,Z 1066.104,A -85,B 0,C 180,E1 15710.638,E2 15710.638} C_VEL
LIN {X 0,Y 358.205,Z 1048.796,A -85,B 0,C 180,E1 15707.471,E2 15707.471} C_VEL
LIN {X 0,Y 365.34,Z 1033.239,A -85,B 0,C 180,E1 15705.08,E2 15705.08} C_VEL
LIN {X 0,Y 373.666,Z 1014.376,A -85,B 0,C 180,E1 15702.619,E2 15702.619} C_VEL
LIN {X 0,Y 381.272,Z 995.817,A -85,B 0,C 180,E1 15700.604,E2 15700.604} C_VEL
LIN {X 0,Y 389.018,Z 975.661,A -85,B 0,C 180,E1 15698.746,E2 15698.746} C_VEL
LIN {X 0,Y 396.356,Z 954.337,A -85,B 0,C 180,E1 15697.138,E2 15697.138} C_VEL
LIN {X 0,Y 403.034,Z 932.839,A -85,B 0,C 180,E1 15695.781,E2 15695.781} C_VEL
LIN {X 0,Y 409.316,Z 909.28,A -85,B 0,C 180,E1 15694.59,E2 15694.59} C_VEL
LIN {X 0,Y 414.521,Z 886.657,A -85,B 0,C 180,E1 15693.675,E2 15693.675} C_VEL
LIN {X 0,Y 419.039,Z 861.962,A -85,B 0,C 180,E1 15692.914,E2 15692.914} C_VEL
LIN {X 0,Y 422.197,Z 839.092,A -85,B 0,C 180,E1 15692.374,E2 15692.374} C_VEL
LIN {X 0,Y 424.926,Z 805.156,A -85,B 0,C 180,E1 15691.77,E2 15691.77} C_VEL
LIN {X 0,Y 439.09,Z 597.321,A -85,B 0,C 180,E1 15688.373,E2 15688.373} C_VEL
LIN {X 0,Y 431.739,Z 583.089,A -85,B 0,C 180,E1 15686.143,E2 15686.143} C_VEL
LIN {X 0,Y 424.483,Z 569.88,A -85,B 0,C 180,E1 15683.717,E2 15683.717} C_VEL
LIN {X 0,Y 417.544,Z 558.135,A -85,B 0,C 180,E1 15681.125,E2 15681.125} C_VEL
LIN {X 0,Y 411.647,Z 548.702,A -85,B 0,C 180,E1 15678.628,E2 15678.628} C_VEL
LIN {X 0,Y 406.682,Z 542.057,A -85,B 0,C 180,E1 15676.277,E2 15676.277} C_VEL
LIN {X 0,Y 403.265,Z 537.444,A -85,B 0,C 180,E1 15674.43,E2 15674.43} C_VEL
LIN {X 0,Y 399.594,Z 532.422,A -85,B 0,C 180,E1 15672.134,E2 15672.134} C_VEL
LIN {X 0,Y 396.348,Z 528.43,A -85,B 0,C 180,E1 15669.731,E2 15669.731} C_VEL
LIN {X 0,Y 395.386,Z 526.885,A -85,B 0,C 180,E1 15668.874,E2 15668.874} C_VEL
LIN {X 0,Y 392.338,Z 523.562,A -85,B 0,C 180,E1 15665.704,E2 15665.704} C_VEL
LIN {X 0,Y 391.257,Z 521.149,A -85,B 0,C 180,E1 15663.957,E2 15663.957} C_VEL
LIN {X 0,Y 389.455,Z 520.147,A -85,B 0,C 180,E1 15657.646,E2 15657.646} C_VEL
LIN {X 0,Y 391.433,Z 521.344,A -85,B 0,C 180,E1 15652.219,E2 15652.219} C_VEL
LIN {X 0,Y 393.273,Z 525.031,A -85,B 0,C 180,E1 15649.6,E2 15649.6} C_VEL
LIN {X 0,Y 395.794,Z 527.383,A -85,B 0,C 180,E1 15647.229,E2 15647.229} C_VEL
LIN {X 0,Y 398.748,Z 531.708,A -85,B 0,C 180,E1 15644.883,E2 15644.883} C_VEL
LIN {X 0,Y 400.226,Z 533.328,A -85,B 0,C 180,E1 15643.9,E2 15643.9} C_VEL
LIN {X 0,Y 404.515,Z 539.095,A -85,B 0,C 180,E1 15641.331,E2 15641.331} C_VEL
LIN {X 0,Y 408.696,Z 544.847,A -85,B 0,C 180,E1 15639.184,E2 15639.184} C_VEL
LIN {X 0,Y 412.97,Z 550.764,A -85,B 0,C 180,E1 15637.245,E2 15637.245} C_VEL
LIN {X 0,Y 418.554,Z 558.685,A -85,B 0,C 180,E1 15634.986,E2 15634.986} C_VEL
LIN {X 0,Y 426.414,Z 570.385,A -85,B 0,C 180,E1 15632.184,E2 15632.184} C_VEL
LIN {X 0,Y 435.125,Z 584.396,A -85,B 0,C 180,E1 15629.441,E2 15629.441} C_VEL
LIN {X 0,Y 439.342,Z 591.673,A -85,B 0,C 180,E1 15628.217,E2 15628.217} C_VEL
LIN {X 0,Y 423.894,Z 813.805,A -85,B 0,C 180,E1 15624.582,E2 15624.582} C_VEL
LIN {X 0,Y 420.843,Z 839.909,A -85,B 0,C 180,E1 15623.992,E2 15623.992} C_VEL
LIN {X 0,Y 417.347,Z 861.416,A -85,B 0,C 180,E1 15623.329,E2 15623.329} C_VEL
LIN {X 0,Y 412.919,Z 883.614,A -85,B 0,C 180,E1 15622.472,E2 15622.472} C_VEL
LIN {X 0,Y 407.51,Z 905.556,A -85,B 0,C 180,E1 15621.398,E2 15621.398} C_VEL
LIN {X 0,Y 401.941,Z 925.338,A -85,B 0,C 180,E1 15620.236,E2 15620.236} C_VEL
LIN {X 0,Y 394.538,Z 948.257,A -85,B 0,C 180,E1 15618.605,E2 15618.605} C_VEL
LIN {X 0,Y 387.982,Z 966.487,A -85,B 0,C 180,E1 15617.047,E2 15617.047} C_VEL
LIN {X 0,Y 379.55,Z 987.842,A -85,B 0,C 180,E1 15614.874,E2 15614.874} C_VEL
LIN {X 0,Y 372.466,Z 1004.348,A -85,B 0,C 180,E1 15612.872,E2 15612.872} C_VEL
LIN {X 0,Y 364.456,Z 1022.063,A -85,B 0,C 180,E1 15610.351,E2 15610.351} C_VEL
LIN {X 0,Y 356.833,Z 1037.875,A -85,B 0,C 180,E1 15607.652,E2 15607.652} C_VEL
LIN {X 0,Y 349.23,Z 1053.386,A -85,B 0,C 180,E1 15604.534,E2 15604.534} C_VEL
LIN {X 0,Y 342.538,Z 1066.654,A -85,B 0,C 180,E1 15601.305,E2 15601.305} C_VEL
LIN {X 0,Y 336.53,Z 1078.859,A -85,B 0,C 180,E1 15597.806,E2 15597.806} C_VEL
LIN {X 0,Y 331.331,Z 1089.625,A -85,B 0,C 180,E1 15594.042,E2 15594.042} C_VEL
LIN {X 0,Y 327.386,Z 1098.453,A -85,B 0,C 180,E1 15590.342,E2 15590.342} C_VEL
LIN {X 0,Y 324.004,Z 1106.883,A -85,B 0,C 180,E1 15585.942,E2 15585.942} C_VEL
LIN {X 0,Y 322.086,Z 1112.565,A -85,B 0,C 180,E1 15582.187,E2 15582.187} C_VEL
LIN {X 0,Y 320.807,Z 1117.555,A -85,B 0,C 180,E1 15577.882,E2 15577.882} C_VEL
LIN {X 0,Y 320.25,Z 1120.631,A -85,B 0,C 180,E1 15573.939,E2 15573.939} C_VEL
LIN {X 0,Y 320.096,Z 1122.298,A -85,B 0,C 180,E1 15570.537,E2 15570.537} C_VEL
LIN {X 0,Y 320.046,Z 1123.078,A -85,B 0,C 180,E1 15566.776,E2 15566.776} C_VEL
LIN {X 0,Y 320.118,Z 1122.535,A -85,B 0,C 180,E1 15562.642,E2 15562.642} C_VEL
LIN {X 0,Y 320.401,Z 1120.911,A -85,B 0,C 180,E1 15559.026,E2 15559.026} C_VEL
LIN {X 0,Y 321.079,Z 1118.08,A -85,B 0,C 180,E1 15555.205,E2 15555.205} C_VEL
LIN {X 0,Y 322.751,Z 1113.064,A -85,B 0,C 180,E1 15550.641,E2 15550.641} C_VEL
LIN {X 0,Y 325.049,Z 1107.402,A -85,B 0,C 180,E1 15546.812,E2 15546.812} C_VEL
LIN {X 0,Y 328.683,Z 1099.707,A -85,B 0,C 180,E1 15542.654,E2 15542.654} C_VEL
LIN {X 0,Y 333.345,Z 1090.521,A -85,B 0,C 180,E1 15538.74,E2 15538.74} C_VEL
LIN {X 0,Y 339.256,Z 1079.733,A -85,B 0,C 180,E1 15534.919,E2 15534.919} C_VEL
LIN {X 0,Y 346.01,Z 1067.405,A -85,B 0,C 180,E1 15531.377,E2 15531.377} C_VEL
LIN {X 0,Y 353.769,Z 1053.499,A -85,B 0,C 180,E1 15528.017,E2 15528.017} C_VEL
LIN {X 0,Y 361.951,Z 1038.225,A -85,B 0,C 180,E1 15524.992,E2 15524.992} C_VEL
LIN {X 0,Y 370.37,Z 1022.125,A -85,B 0,C 180,E1 15522.292,E2 15522.292} C_VEL
LIN {X 0,Y 378.959,Z 1004.491,A -85,B 0,C 180,E1 15519.842,E2 15519.842} C_VEL
LIN {X 0,Y 387.234,Z 986.544,A -85,B 0,C 180,E1 15517.732,E2 15517.732} C_VEL
LIN {X 0,Y 395.613,Z 966.558,A -85,B 0,C 180,E1 15515.775,E2 15515.775} C_VEL
LIN {X 0,Y 402.751,Z 947.916,A -85,B 0,C 180,E1 15514.236,E2 15514.236} C_VEL
LIN {X 0,Y 403.244,Z 946.599,A -85,B 0,C 180,E1 15514.135,E2 15514.135} C_VEL
LIN {X 0,Y 404.979,Z 940.255,A -85,B 0,C 180,E1 15513.548,E2 15513.548} C_VEL
LIN {X 0,Y 407.045,Z 923.578,A -85,B 0,C 180,E1 15511.719,E2 15511.719} C_VEL
LIN {X 0,Y 408.469,Z 917.861,A -85,B 0,C 180,E1 15511.288,E2 15511.288} C_VEL
LIN {X 0,Y 414.946,Z 895.161,A -85,B 0,C 180,E1 15510.108,E2 15510.108} C_VEL
LIN {X 0,Y 419.979,Z 874.311,A -85,B 0,C 180,E1 15509.227,E2 15509.227} C_VEL
LIN {X 0,Y 424.947,Z 849.058,A -85,B 0,C 180,E1 15508.391,E2 15508.391} C_VEL
LIN {X 0,Y 428.238,Z 826.711,A -85,B 0,C 180,E1 15507.836,E2 15507.836} C_VEL
LIN {X 0,Y 430.921,Z 799.465,A -85,B 0,C 180,E1 15507.334,E2 15507.334} C_VEL
LIN {X 0,Y 445.701,Z 602.946,A -85,B 0,C 180,E1 15504.186,E2 15504.186} C_VEL
LIN {X 0,Y 438.552,Z 591.083,A -85,B 0,C 180,E1 15501.676,E2 15501.676} C_VEL
LIN {X 0,Y 431.656,Z 580.431,A -85,B 0,C 180,E1 15498.923,E2 15498.923} C_VEL
LIN {X 0,Y 426.761,Z 573.2,A -85,B 0,C 180,E1 15496.679,E2 15496.679} C_VEL
LIN {X 0,Y 423.482,Z 568.467,A -85,B 0,C 180,E1 15494.984,E2 15494.984} C_VEL
LIN {X 0,Y 420.851,Z 564.657,A -85,B 0,C 180,E1 15493.464,E2 15493.464} C_VEL
LIN {X 0,Y 417.807,Z 560.246,A -85,B 0,C 180,E1 15491.457,E2 15491.457} C_VEL
LIN {X 0,Y 414.802,Z 556.018,A -85,B 0,C 180,E1 15489.084,E2 15489.084} C_VEL
LIN {X 0,Y 413.973,Z 554.964,A -85,B 0,C 180,E1 15488.333,E2 15488.333} C_VEL
LIN {X 0,Y 411.264,Z 551.23,A -85,B 0,C 180,E1 15485.231,E2 15485.231} C_VEL
LIN {X 0,Y 410.663,Z 549.741,A -85,B 0,C 180,E1 15484.189,E2 15484.189} C_VEL
LIN {X 0,Y 408.933,Z 548.645,A -85,B 0,C 180,E1 15478.459,E2 15478.459} C_VEL
LIN {X 0,Y 410.82,Z 549.975,A -85,B 0,C 180,E1 15473.01,E2 15473.01} C_VEL
LIN {X 0,Y 412.969,Z 553.956,A -85,B 0,C 180,E1 15470.101,E2 15470.101} C_VEL
LIN {X 0,Y 414.727,Z 555.801,A -85,B 0,C 180,E1 15468.457,E2 15468.457} C_VEL
LIN {X 0,Y 417.803,Z 560.192,A -85,B 0,C 180,E1 15466.012,E2 15466.012} C_VEL
LIN {X 0,Y 422.43,Z 566.842,A -85,B 0,C 180,E1 15463.074,E2 15463.074} C_VEL
LIN {X 0,Y 426.623,Z 573.778,A -85,B 0,C 180,E1 15460.809,E2 15460.809} C_VEL
LIN {X 0,Y 432.154,Z 583.144,A -85,B 0,C 180,E1 15458.236,E2 15458.236} C_VEL
LIN {X 0,Y 439.231,Z 596.092,A -85,B 0,C 180,E1 15455.38,E2 15455.38} C_VEL
LIN {X 0,Y 445.51,Z 608.272,A -85,B 0,C 180,E1 15453.139,E2 15453.139} C_VEL
LIN {X 0,Y 429.28,Z 824.121,A -85,B 0,C 180,E1 15449.657,E2 15449.657} C_VEL
LIN {X 0,Y 426.781,Z 846.411,A -85,B 0,C 180,E1 15449.224,E2 15449.224} C_VEL
LIN {X 0,Y 422.296,Z 873.028,A -85,B 0,C 180,E1 15448.554,E2 15448.554} C_VEL
LIN {X 0,Y 417.7,Z 893.997,A -85,B 0,C 180,E1 15447.866,E2 15447.866} C_VEL
LIN {X 0,Y 411.381,Z 918.105,A -85,B 0,C 180,E1 15446.86,E2 15446.86} C_VEL
LIN {X 0,Y 405.058,Z 938.56,A -85,B 0,C 180,E1 15445.787,E2 15445.787} C_VEL
LIN {X 0,Y 397.357,Z 960.848,A -85,B 0,C 180,E1 15444.369,E2 15444.369} C_VEL
LIN {X 0,Y 389.278,Z 981.263,A -85,B 0,C 180,E1 15442.775,E2 15442.775} C_VEL
LIN {X 0,Y 380.934,Z 1000.814,A -85,B 0,C 180,E1 15440.953,E2 15440.953} C_VEL
LIN {X 0,Y 371.748,Z 1020.38,A -85,B 0,C 180,E1 15438.744,E2 15438.744} C_VEL
LIN {X 0,Y 363.36,Z 1037.282,A -85,B 0,C 180,E1 15436.477,E2 15436.477} C_VEL
LIN {X 0,Y 354.398,Z 1054.383,A -85,B 0,C 180,E1 15433.728,E2 15433.728} C_VEL
LIN {X 0,Y 346.892,Z 1068.243,A -85,B 0,C 180,E1 15431.086,E2 15431.086} C_VEL
LIN {X 0,Y 338.64,Z 1083.317,A -85,B 0,C 180,E1 15427.677,E2 15427.677} C_VEL
LIN {X 0,Y 331.835,Z 1095.669,A -85,B 0,C 180,E1 15424.296,E2 15424.296} C_VEL
LIN {X 0,Y 325.609,Z 1107.526,A -85,B 0,C 180,E1 15420.444,E2 15420.444} C_VEL
LIN {X 0,Y 320.654,Z 1117.407,A -85,B 0,C 180,E1 15416.482,E2 15416.482} C_VEL
LIN {X 0,Y 316.806,Z 1126.145,A -85,B 0,C 180,E1 15412.256,E2 15412.256} C_VEL
LIN {X 0,Y 314.138,Z 1133.331,A -85,B 0,C 180,E1 15407.792,E2 15407.792} C_VEL
LIN {X 0,Y 312.78,Z 1138.27,A -85,B 0,C 180,E1 15403.872,E2 15403.872} C_VEL
LIN {X 0,Y 312.083,Z 1142.477,A -85,B 0,C 180,E1 15399.218,E2 15399.218} C_VEL
LIN {X 0,Y 311.987,Z 1144.523,A -85,B 0,C 180,E1 15395.517,E2 15395.517} C_VEL
LIN {X 0,Y 312.035,Z 1145.422,A -85,B 0,C 180,E1 15392.204,E2 15392.204} C_VEL
LIN {X 0,Y 312.053,Z 1145.407,A -85,B 0,C 180,E1 15388.898,E2 15388.898} C_VEL
LIN {X 0,Y 312.007,Z 1144.333,A -85,B 0,C 180,E1 15385.22,E2 15385.22} C_VEL
LIN {X 0,Y 312.079,Z 1141.654,A -85,B 0,C 180,E1 15380.967,E2 15380.967} C_VEL
LIN {X 0,Y 312.549,Z 1137.816,A -85,B 0,C 180,E1 15377.059,E2 15377.059} C_VEL
LIN {X 0,Y 313.675,Z 1132.722,A -85,B 0,C 180,E1 15373.137,E2 15373.137} C_VEL
LIN {X 0,Y 316.12,Z 1124.811,A -85,B 0,C 180,E1 15368.475,E2 15368.475} C_VEL
LIN {X 0,Y 319.088,Z 1117.013,A -85,B 0,C 180,E1 15364.775,E2 15364.775} C_VEL
LIN {X 0,Y 323.796,Z 1106.237,A -85,B 0,C 180,E1 15360.555,E2 15360.555} C_VEL
LIN {X 0,Y 328.923,Z 1095.314,A -85,B 0,C 180,E1 15357.034,E2 15357.034} C_VEL
LIN {X 0,Y 335.497,Z 1082.048,A -85,B 0,C 180,E1 15353.411,E2 15353.411} C_VEL
LIN {X 0,Y 342.775,Z 1067.321,A -85,B 0,C 180,E1 15350.102,E2 15350.102} C_VEL
LIN {X 0,Y 350.74,Z 1051.3,A -85,B 0,C 180,E1 15347.051,E2 15347.051} C_VEL
LIN {X 0,Y 358.704,Z 1034.493,A -85,B 0,C 180,E1 15344.4,E2 15344.4} C_VEL
LIN {X 0,Y 366.817,Z 1016.812,A -85,B 0,C 180,E1 15342.03,E2 15342.03} C_VEL
LIN {X 0,Y 375.13,Z 997.299,A -85,B 0,C 180,E1 15339.856,E2 15339.856} C_VEL
LIN {X 0,Y 382.497,Z 978.72,A -85,B 0,C 180,E1 15338.108,E2 15338.108} C_VEL
LIN {X 0,Y 390.553,Z 956.43,A -85,B 0,C 180,E1 15336.372,E2 15336.372} C_VEL
LIN {X 0,Y 396.734,Z 937.246,A -85,B 0,C 180,E1 15335.131,E2 15335.131} C_VEL
LIN {X 0,Y 403.313,Z 914.292,A -85,B 0,C 180,E1 15333.905,E2 15333.905} C_VEL
LIN {X 0,Y 408.581,Z 892.506,A -85,B 0,C 180,E1 15332.986,E2 15332.986} C_VEL
LIN {X 0,Y 413.125,Z 870.353,A -85,B 0,C 180,E1 15332.239,E2 15332.239} C_VEL
LIN {X 0,Y 416.955,Z 845.438,A -85,B 0,C 180,E1 15331.603,E2 15331.603} C_VEL
LIN {X 0,Y 419.322,Z 822.507,A -85,B 0,C 180,E1 15331.149,E2 15331.149} C_VEL
LIN {X 0,Y 434.82,Z 601.742,A -85,B 0,C 180,E1 15327.53,E2 15327.53} C_VEL
LIN {X 0,Y 434.519,Z 600.596,A -85,B 0,C 180,E1 15327.421,E2 15327.421} C_VEL
LIN {X 0,Y 427.047,Z 585.98,A -85,B 0,C 180,E1 15325.03,E2 15325.03} C_VEL
LIN {X 0,Y 418.999,Z 571.412,A -85,B 0,C 180,E1 15322.151,E2 15322.151} C_VEL
LIN {X 0,Y 412.27,Z 560.082,A -85,B 0,C 180,E1 15319.407,E2 15319.407} C_VEL
LIN {X 0,Y 408.588,Z 554.518,A -85,B 0,C 180,E1 15317.739,E2 15317.739} C_VEL
LIN {X 0,Y 404.762,Z 549.268,A -85,B 0,C 180,E1 15315.841,E2 15315.841} C_VEL
LIN {X 0,Y 401.798,Z 545.125,A -85,B 0,C 180,E1 15314.189,E2 15314.189} C_VEL
LIN {X 0,Y 397.981,Z 539.938,A -85,B 0,C 180,E1 15311.742,E2 15311.742} C_VEL
LIN {X 0,Y 394.789,Z 535.666,A -85,B 0,C 180,E1 15309.255,E2 15309.255} C_VEL
LIN {X 0,Y 394.08,Z 534.649,A -85,B 0,C 180,E1 15308.61,E2 15308.61} C_VEL
LIN {X 0,Y 391.142,Z 531.257,A -85,B 0,C 180,E1 15305.427,E2 15305.427} C_VEL
LIN {X 0,Y 390.19,Z 529.048,A -85,B 0,C 180,E1 15303.82,E2 15303.82} C_VEL
LIN {X 0,Y 388.49,Z 528.098,A -85,B 0,C 180,E1 15297.492,E2 15297.492} C_VEL
LIN {X 0,Y 390.362,Z 529.294,A -85,B 0,C 180,E1 15292.346,E2 15292.346} C_VEL
LIN {X 0,Y 392.302,Z 533.069,A -85,B 0,C 180,E1 15289.574,E2 15289.574} C_VEL
LIN {X 0,Y 394.568,Z 535.254,A -85,B 0,C 180,E1 15287.412,E2 15287.412} C_VEL
LIN {X 0,Y 397.581,Z 539.614,A -85,B 0,C 180,E1 15284.987,E2 15284.987} C_VEL
LIN {X 0,Y 398.923,Z 541.241,A -85,B 0,C 180,E1 15284.07,E2 15284.07} C_VEL
LIN {X 0,Y 402.916,Z 546.662,A -85,B 0,C 180,E1 15281.629,E2 15281.629} C_VEL
LIN {X 0,Y 406.949,Z 552.324,A -85,B 0,C 180,E1 15279.505,E2 15279.505} C_VEL
LIN {X 0,Y 411.682,Z 558.98,A -85,B 0,C 180,E1 15277.321,E2 15277.321} C_VEL
LIN {X 0,Y 418.936,Z 569.574,A -85,B 0,C 180,E1 15274.405,E2 15274.405} C_VEL
LIN {X 0,Y 427.103,Z 582.406,A -85,B 0,C 180,E1 15271.548,E2 15271.548} C_VEL
LIN {X 0,Y 435.101,Z 595.802,A -85,B 0,C 180,E1 15269.065,E2 15269.065} C_VEL
LIN {X 0,Y 419.466,Z 814.489,A -85,B 0,C 180,E1 15265.482,E2 15265.482} C_VEL
LIN {X 0,Y 416.208,Z 841.274,A -85,B 0,C 180,E1 15264.872,E2 15264.872} C_VEL
LIN {X 0,Y 412.657,Z 862.492,A -85,B 0,C 180,E1 15264.213,E2 15264.213} C_VEL
LIN {X 0,Y 407.638,Z 886.47,A -85,B 0,C 180,E1 15263.266,E2 15263.266} C_VEL
LIN {X 0,Y 402.288,Z 907.471,A -85,B 0,C 180,E1 15262.223,E2 15262.223} C_VEL
LIN {X 0,Y 395.714,Z 929.972,A -85,B 0,C 180,E1 15260.871,E2 15260.871} C_VEL
LIN {X 0,Y 388.725,Z 950.511,A -85,B 0,C 180,E1 15259.36,E2 15259.36} C_VEL
LIN {X 0,Y 381.422,Z 970.155,A -85,B 0,C 180,E1 15257.645,E2 15257.645} C_VEL
LIN {X 0,Y 373.211,Z 989.989,A -85,B 0,C 180,E1 15255.561,E2 15255.561} C_VEL
LIN {X 0,Y 365.902,Z 1006.46,A -85,B 0,C 180,E1 15253.522,E2 15253.522} C_VEL
LIN {X 0,Y 356.968,Z 1025.29,A -85,B 0,C 180,E1 15250.742,E2 15250.742} C_VEL
LIN {X 0,Y 349.595,Z 1040.091,A -85,B 0,C 180,E1 15248.136,E2 15248.136} C_VEL
LIN {X 0,Y 341.478,Z 1055.896,A -85,B 0,C 180,E1 15244.819,E2 15244.819} C_VEL
LIN {X 0,Y 334.992,Z 1068.334,A -85,B 0,C 180,E1 15241.691,E2 15241.691} C_VEL
LIN {X 0,Y 328.297,Z 1081.338,A -85,B 0,C 180,E1 15237.774,E2 15237.774} C_VEL
LIN {X 0,Y 323.433,Z 1091.056,A -85,B 0,C 180,E1 15234.218,E2 15234.218} C_VEL
LIN {X 0,Y 319.171,Z 1100.317,A -85,B 0,C 180,E1 15230.158,E2 15230.158} C_VEL
LIN {X 0,Y 316.008,Z 1107.832,A -85,B 0,C 180,E1 15225.979,E2 15225.979} C_VEL
LIN {X 0,Y 313.996,Z 1113.653,A -85,B 0,C 180,E1 15221.946,E2 15221.946} C_VEL
LIN {X 0,Y 312.747,Z 1118.341,A -85,B 0,C 180,E1 15217.532,E2 15217.532} C_VEL
LIN {X 0,Y 312.251,Z 1121.053,A -85,B 0,C 180,E1 15213.856,E2 15213.856} C_VEL
LIN {X 0,Y 312.108,Z 1122.731,A -85,B 0,C 180,E1 15210.184,E2 15210.184} C_VEL
LIN {X 0,Y 312.057,Z 1123.384,A -85,B 0,C 180,E1 15205.958,E2 15205.958} C_VEL
LIN {X 0,Y 312.16,Z 1122.675,A -85,B 0,C 180,E1 15202.083,E2 15202.083} C_VEL
LIN {X 0,Y 312.491,Z 1120.954,A -85,B 0,C 180,E1 15198.37,E2 15198.37} C_VEL
LIN {X 0,Y 313.472,Z 1117.527,A -85,B 0,C 180,E1 15193.888,E2 15193.888} C_VEL
LIN {X 0,Y 315.293,Z 1112.55,A -85,B 0,C 180,E1 15189.583,E2 15189.583} C_VEL
LIN {X 0,Y 318.204,Z 1106.139,A -85,B 0,C 180,E1 15185.296,E2 15185.296} C_VEL
LIN {X 0,Y 322.426,Z 1097.755,A -85,B 0,C 180,E1 15180.989,E2 15180.989} C_VEL
LIN {X 0,Y 327.303,Z 1088.893,A -85,B 0,C 180,E1 15177.267,E2 15177.267} C_VEL
LIN {X 0,Y 334.041,Z 1077.059,A -85,B 0,C 180,E1 15173.226,E2 15173.226} C_VEL
LIN {X 0,Y 340.658,Z 1065.657,A -85,B 0,C 180,E1 15169.999,E2 15169.999} C_VEL
LIN {X 0,Y 349.451,Z 1050.298,A -85,B 0,C 180,E1 15166.403,E2 15166.403} C_VEL
LIN {X 0,Y 357.058,Z 1036.632,A -85,B 0,C 180,E1 15163.739,E2 15163.739} C_VEL
LIN {X 0,Y 366.62,Z 1018.683,A -85,B 0,C 180,E1 15160.814,E2 15160.814} C_VEL
LIN {X 0,Y 374.545,Z 1002.855,A -85,B 0,C 180,E1 15158.66,E2 15158.66} C_VEL
LIN {X 0,Y 383.437,Z 983.946,A -85,B 0,C 180,E1 15156.481,E2 15156.481} C_VEL
LIN {X 0,Y 391.479,Z 965.031,A -85,B 0,C 180,E1 15154.671,E2 15154.671} C_VEL
LIN {X 0,Y 399.469,Z 944.568,A -85,B 0,C 180,E1 15153.015,E2 15153.015} C_VEL
LIN {X 0,Y 406.804,Z 923.011,A -85,B 0,C 180,E1 15151.592,E2 15151.592} C_VEL
LIN {X 0,Y 408.469,Z 917.861,A -85,B 0,C 180,E1 15151.288,E2 15151.288} C_VEL
LIN {X 0,Y 410.034,Z 911.142,A -85,B 0,C 180,E1 15150.789,E2 15150.789} C_VEL
LIN {X 0,Y 411.69,Z 893.499,A -85,B 0,C 180,E1 15149.162,E2 15149.162} C_VEL
LIN {X 0,Y 412.878,Z 887.506,A -85,B 0,C 180,E1 15148.8,E2 15148.8} C_VEL
LIN {X 0,Y 418.369,Z 863.285,A -85,B 0,C 180,E1 15147.883,E2 15147.883} C_VEL
LIN {X 0,Y 422.119,Z 842.602,A -85,B 0,C 180,E1 15147.268,E2 15147.268} C_VEL
LIN {X 0,Y 425.599,Z 816.536,A -85,B 0,C 180,E1 15146.686,E2 15146.686} C_VEL
LIN {X 0,Y 434.859,Z 698.197,A -85,B 0,C 180,E1 15144.765,E2 15144.765} C_VEL
LIN {X 0,Y 441.936,Z 607.625,A -85,B 0,C 180,E1 15143.325,E2 15143.325} C_VEL
LIN {X 0,Y 435.728,Z 597.19,A -85,B 0,C 180,E1 15141.047,E2 15141.047} C_VEL
LIN {X 0,Y 428.919,Z 586.383,A -85,B 0,C 180,E1 15138.203,E2 15138.203} C_VEL
LIN {X 0,Y 422.86,Z 577.292,A -85,B 0,C 180,E1 15135.217,E2 15135.217} C_VEL
LIN {X 0,Y 419.209,Z 572.067,A -85,B 0,C 180,E1 15133.097,E2 15133.097} C_VEL
LIN {X 0,Y 416.441,Z 567.945,A -85,B 0,C 180,E1 15131.215,E2 15131.215} C_VEL
LIN {X 0,Y 413.443,Z 563.557,A -85,B 0,C 180,E1 15128.764,E2 15128.764} C_VEL
LIN {X 0,Y 410.059,Z 558.819,A -85,B 0,C 180,E1 15124.896,E2 15124.896} C_VEL
LIN {X 0,Y 409.512,Z 557.612,A -85,B 0,C 180,E1 15123.92,E2 15123.92} C_VEL
LIN {X 0,Y 407.964,Z 556.589,A -85,B 0,C 180,E1 15118.315,E2 15118.315} C_VEL
LIN {X 0,Y 409.753,Z 557.906,A -85,B 0,C 180,E1 15113.133,E2 15113.133} C_VEL
LIN {X 0,Y 411.998,Z 561.985,A -85,B 0,C 180,E1 15110.078,E2 15110.078} C_VEL
LIN {X 0,Y 413.515,Z 563.649,A -85,B 0,C 180,E1 15108.634,E2 15108.634} C_VEL
LIN {X 0,Y 417.292,Z 569.187,A -85,B 0,C 180,E1 15105.641,E2 15105.641} C_VEL
LIN {X 0,Y 420.982,Z 574.577,A -85,B 0,C 180,E1 15103.298,E2 15103.298} C_VEL
LIN {X 0,Y 424.974,Z 581.377,A -85,B 0,C 180,E1 15101.089,E2 15101.089} C_VEL
LIN {X 0,Y 430.185,Z 590.454,A -85,B 0,C 180,E1 15098.597,E2 15098.597} C_VEL
LIN {X 0,Y 436.879,Z 602.984,A -85,B 0,C 180,E1 15095.815,E2 15095.815} C_VEL
LIN {X 0,Y 441.737,Z 612.79,A -85,B 0,C 180,E1 15094.002,E2 15094.002} C_VEL
LIN {X 0,Y 424.979,Z 828.775,A -85,B 0,C 180,E1 15090.517,E2 15090.517} C_VEL
LIN {X 0,Y 421.64,Z 854.547,A -85,B 0,C 180,E1 15089.986,E2 15089.986} C_VEL
LIN {X 0,Y 417.509,Z 876.659,A -85,B 0,C 180,E1 15089.392,E2 15089.392} C_VEL
LIN {X 0,Y 412.282,Z 899.438,A -85,B 0,C 180,E1 15088.616,E2 15088.616} C_VEL
LIN {X 0,Y 406.014,Z 921.641,A -85,B 0,C 180,E1 15087.641,E2 15087.641} C_VEL
LIN {X 0,Y 399.585,Z 941.675,A -85,B 0,C 180,E1 15086.567,E2 15086.567} C_VEL
LIN {X 0,Y 391.076,Z 964.932,A -85,B 0,C 180,E1 15085.03,E2 15085.03} C_VEL
LIN {X 0,Y 383.458,Z 983.537,A -85,B 0,C 180,E1 15083.543,E2 15083.543} C_VEL
LIN {X 0,Y 374.15,Z 1004.374,A -85,B 0,C 180,E1 15081.539,E2 15081.539} C_VEL
LIN {X 0,Y 365.566,Z 1021.975,A -85,B 0,C 180,E1 15079.498,E2 15079.498} C_VEL
LIN {X 0,Y 356.193,Z 1040.176,A -85,B 0,C 180,E1 15076.989,E2 15076.989} C_VEL
LIN {X 0,Y 347.534,Z 1055.955,A -85,B 0,C 180,E1 15074.358,E2 15074.358} C_VEL
LIN {X 0,Y 338.993,Z 1071.204,A -85,B 0,C 180,E1 15071.354,E2 15071.354} C_VEL
LIN {X 0,Y 330.599,Z 1085.73,A -85,B 0,C 180,E1 15067.871,E2 15067.871} C_VEL
LIN {X 0,Y 323.737,Z 1097.807,A -85,B 0,C 180,E1 15064.417,E2 15064.417} C_VEL
LIN {X 0,Y 317.085,Z 1109.815,A -85,B 0,C 180,E1 15060.228,E2 15060.228} C_VEL
LIN {X 0,Y 312.36,Z 1119.038,A -85,B 0,C 180,E1 15056.323,E2 15056.323} C_VEL
LIN {X 0,Y 308.34,Z 1127.834,A -85,B 0,C 180,E1 15051.696,E2 15051.696} C_VEL
LIN {X 0,Y 306.066,Z 1133.871,A -85,B 0,C 180,E1 15047.687,E2 15047.687} C_VEL
LIN {X 0,Y 304.59,Z 1139.235,A -85,B 0,C 180,E1 15043.092,E2 15043.092} C_VEL
LIN {X 0,Y 304.07,Z 1142.567,A -85,B 0,C 180,E1 15038.891,E2 15038.891} C_VEL
LIN {X 0,Y 303.99,Z 1144.322,A -85,B 0,C 180,E1 15035.474,E2 15035.474} C_VEL
LIN {X 0,Y 304.043,Z 1145.166,A -85,B 0,C 180,E1 15032.073,E2 15032.073} C_VEL
LIN {X 0,Y 304.058,Z 1145.073,A -85,B 0,C 180,E1 15028.492,E2 15028.492} C_VEL
LIN {X 0,Y 304.006,Z 1143.722,A -85,B 0,C 180,E1 15024.337,E2 15024.337} C_VEL
LIN {X 0,Y 304.14,Z 1140.842,A -85,B 0,C 180,E1 15020.157,E2 15020.157} C_VEL
LIN {X 0,Y 304.7,Z 1137.06,A -85,B 0,C 180,E1 15016.333,E2 15016.333} C_VEL
LIN {X 0,Y 306.189,Z 1131.2,A -85,B 0,C 180,E1 15011.859,E2 15011.859} C_VEL
LIN {X 0,Y 308.717,Z 1123.721,A -85,B 0,C 180,E1 15007.531,E2 15007.531} C_VEL
LIN {X 0,Y 312.377,Z 1114.974,A -85,B 0,C 180,E1 15003.376,E2 15003.376} C_VEL
LIN {X 0,Y 317.287,Z 1104.359,A -85,B 0,C 180,E1 14999.301,E2 14999.301} C_VEL
LIN {X 0,Y 322.615,Z 1093.647,A -85,B 0,C 180,E1 14995.845,E2 14995.845} C_VEL
LIN {X 0,Y 330.291,Z 1078.749,A -85,B 0,C 180,E1 14991.861,E2 14991.861} C_VEL
LIN {X 0,Y 337.294,Z 1065.227,A -85,B 0,C 180,E1 14988.849,E2 14988.849} C_VEL
LIN {X 0,Y 346.299,Z 1047.523,A -85,B 0,C 180,E1 14985.558,E2 14985.558} C_VEL
LIN {X 0,Y 354.028,Z 1031.786,A -85,B 0,C 180,E1 14983.117,E2 14983.117} C_VEL
LIN {X 0,Y 363.231,Z 1012.075,A -85,B 0,C 180,E1 14980.556,E2 14980.556} C_VEL
LIN {X 0,Y 370.765,Z 994.707,A -85,B 0,C 180,E1 14978.672,E2 14978.672} C_VEL
LIN {X 0,Y 379.124,Z 974.028,A -85,B 0,C 180,E1 14976.776,E2 14976.776} C_VEL
LIN {X 0,Y 386.699,Z 953.049,A -85,B 0,C 180,E1 14975.206,E2 14975.206} C_VEL
LIN {X 0,Y 393.723,Z 931.474,A -85,B 0,C 180,E1 14973.855,E2 14973.855} C_VEL
LIN {X 0,Y 399.973,Z 908.997,A -85,B 0,C 180,E1 14972.731,E2 14972.731} C_VEL
LIN {X 0,Y 405.233,Z 887.166,A -85,B 0,C 180,E1 14971.851,E2 14971.851} C_VEL
LIN {X 0,Y 410.088,Z 862.045,A -85,B 0,C 180,E1 14971.076,E2 14971.076} C_VEL
LIN {X 0,Y 413.333,Z 839.692,A -85,B 0,C 180,E1 14970.548,E2 14970.548} C_VEL
LIN {X 0,Y 416.205,Z 806.692,A -85,B 0,C 180,E1 14969.953,E2 14969.953} C_VEL
LIN {X 0,Y 430.688,Z 605.276,A -85,B 0,C 180,E1 14966.651,E2 14966.651} C_VEL
LIN {X 0,Y 423.517,Z 591.024,A -85,B 0,C 180,E1 14964.255,E2 14964.255} C_VEL
LIN {X 0,Y 415.715,Z 576.655,A -85,B 0,C 180,E1 14961.333,E2 14961.333} C_VEL
LIN {X 0,Y 408.74,Z 564.767,A -85,B 0,C 180,E1 14958.321,E2 14958.321} C_VEL
LIN {X 0,Y 403.382,Z 557.124,A -85,B 0,C 180,E1 14955.675,E2 14955.675} C_VEL
LIN {X 0,Y 400.101,Z 552.551,A -85,B 0,C 180,E1 14953.808,E2 14953.808} C_VEL
LIN {X 0,Y 396.593,Z 547.636,A -85,B 0,C 180,E1 14951.489,E2 14951.489} C_VEL
LIN {X 0,Y 393.48,Z 543.353,A -85,B 0,C 180,E1 14948.991,E2 14948.991} C_VEL
LIN {X 0,Y 392.623,Z 542.289,A -85,B 0,C 180,E1 14948.199,E2 14948.199} C_VEL
LIN {X 0,Y 389.815,Z 538.647,A -85,B 0,C 180,E1 14944.929,E2 14944.929} C_VEL
LIN {X 0,Y 389.126,Z 536.948,A -85,B 0,C 180,E1 14943.683,E2 14943.683} C_VEL
LIN {X 0,Y 387.516,Z 536.039,A -85,B 0,C 180,E1 14937.486,E2 14937.486} C_VEL
LIN {X 0,Y 389.293,Z 537.239,A -85,B 0,C 180,E1 14932.473,E2 14932.473} C_VEL
LIN {X 0,Y 391.2,Z 540.954,A -85,B 0,C 180,E1 14929.693,E2 14929.693} C_VEL
LIN {X 0,Y 393.346,Z 543.117,A -85,B 0,C 180,E1 14927.596,E2 14927.596} C_VEL
LIN {X 0,Y 396.415,Z 547.517,A -85,B 0,C 180,E1 14925.091,E2 14925.091} C_VEL
LIN {X 0,Y 397.626,Z 549.142,A -85,B 0,C 180,E1 14924.241,E2 14924.241} C_VEL
LIN {X 0,Y 401.445,Z 554.42,A -85,B 0,C 180,E1 14921.86,E2 14921.86} C_VEL
LIN {X 0,Y 405.349,Z 560.004,A -85,B 0,C 180,E1 14919.759,E2 14919.759} C_VEL
LIN {X 0,Y 410.705,Z 567.6,A -85,B 0,C 180,E1 14917.264,E2 14917.264} C_VEL
LIN {X 0,Y 418.891,Z 580.078,A -85,B 0,C 180,E1 14913.985,E2 14913.985} C_VEL
LIN {X 0,Y 427.138,Z 593.581,A -85,B 0,C 180,E1 14911.131,E2 14911.131} C_VEL
LIN {X 0,Y 430.93,Z 600.298,A -85,B 0,C 180,E1 14909.924,E2 14909.924} C_VEL
LIN {X 0,Y 415.135,Z 815.266,A -85,B 0,C 180,E1 14906.4,E2 14906.4} C_VEL
LIN {X 0,Y 411.799,Z 841.861,A -85,B 0,C 180,E1 14905.792,E2 14905.792} C_VEL
LIN {X 0,Y 408.168,Z 863.03,A -85,B 0,C 180,E1 14905.135,E2 14905.135} C_VEL
LIN {X 0,Y 403.109,Z 886.644,A -85,B 0,C 180,E1 14904.205,E2 14904.205} C_VEL
LIN {X 0,Y 397.766,Z 907.159,A -85,B 0,C 180,E1 14903.191,E2 14903.191} C_VEL
LIN {X 0,Y 391.33,Z 928.806,A -85,B 0,C 180,E1 14901.904,E2 14901.904} C_VEL
LIN {X 0,Y 383.967,Z 950.056,A -85,B 0,C 180,E1 14900.356,E2 14900.356} C_VEL
LIN {X 0,Y 376.68,Z 969.18,A -85,B 0,C 180,E1 14898.696,E2 14898.696} C_VEL
LIN {X 0,Y 368.166,Z 989.339,A -85,B 0,C 180,E1 14896.598,E2 14896.598} C_VEL
LIN {X 0,Y 360.601,Z 1005.916,A -85,B 0,C 180,E1 14894.55,E2 14894.55} C_VEL
LIN {X 0,Y 351.358,Z 1024.885,A -85,B 0,C 180,E1 14891.753,E2 14891.753} C_VEL
LIN {X 0,Y 343.739,Z 1039.674,A -85,B 0,C 180,E1 14889.141,E2 14889.141} C_VEL
LIN {X 0,Y 335.615,Z 1054.978,A -85,B 0,C 180,E1 14885.939,E2 14885.939} C_VEL
LIN {X 0,Y 328.783,Z 1067.532,A -85,B 0,C 180,E1 14882.774,E2 14882.774} C_VEL
LIN {X 0,Y 322.265,Z 1079.709,A -85,B 0,C 180,E1 14879.152,E2 14879.152} C_VEL
LIN {X 0,Y 316.581,Z 1090.42,A -85,B 0,C 180,E1 14875.238,E2 14875.238} C_VEL
LIN {X 0,Y 312.27,Z 1099.151,A -85,B 0,C 180,E1 14871.409,E2 14871.409} C_VEL
LIN {X 0,Y 308.621,Z 1107.308,A -85,B 0,C 180,E1 14866.953,E2 14866.953} C_VEL
LIN {X 0,Y 306.448,Z 1113.013,A -85,B 0,C 180,E1 14863.011,E2 14863.011} C_VEL
LIN {X 0,Y 304.948,Z 1118.048,A -85,B 0,C 180,E1 14858.485,E2 14858.485} C_VEL
LIN {X 0,Y 304.301,Z 1121.145,A -85,B 0,C 180,E1 14854.334,E2 14854.334} C_VEL
LIN {X 0,Y 304.103,Z 1122.833,A -85,B 0,C 180,E1 14850.754,E2 14850.754} C_VEL
LIN {X 0,Y 304.055,Z 1123.611,A -85,B 0,C 180,E1 14846.984,E2 14846.984} C_VEL
LIN {X 0,Y 304.132,Z 1123.206,A -85,B 0,C 180,E1 14842.633,E2 14842.633} C_VEL
LIN {X 0,Y 304.465,Z 1121.543,A -85,B 0,C 180,E1 14838.636,E2 14838.636} C_VEL
LIN {X 0,Y 305.2,Z 1118.893,A -85,B 0,C 180,E1 14834.806,E2 14834.806} C_VEL
LIN {X 0,Y 306.968,Z 1114.271,A -85,B 0,C 180,E1 14830.198,E2 14830.198} C_VEL
LIN {X 0,Y 309.61,Z 1108.437,A -85,B 0,C 180,E1 14825.988,E2 14825.988} C_VEL
LIN {X 0,Y 313.612,Z 1100.865,A -85,B 0,C 180,E1 14821.637,E2 14821.637} C_VEL
LIN {X 0,Y 318.703,Z 1091.795,A -85,B 0,C 180,E1 14817.555,E2 14817.555} C_VEL
LIN {X 0,Y 324.477,Z 1082.117,A -85,B 0,C 180,E1 14813.944,E2 14813.944} C_VEL
LIN {X 0,Y 332.039,Z 1069.58,A -85,B 0,C 180,E1 14810.102,E2 14810.102} C_VEL
LIN {X 0,Y 339.163,Z 1057.7,A -85,B 0,C 180,E1 14807.077,E2 14807.077} C_VEL
LIN {X 0,Y 348.061,Z 1042.62,A -85,B 0,C 180,E1 14803.858,E2 14803.858} C_VEL
LIN {X 0,Y 356.351,Z 1027.813,A -85,B 0,C 180,E1 14801.237,E2 14801.237} C_VEL
LIN {X 0,Y 365.319,Z 1011.145,A -85,B 0,C 180,E1 14798.734,E2 14798.734} C_VEL
LIN {X 0,Y 374.304,Z 992.993,A -85,B 0,C 180,E1 14796.479,E2 14796.479} C_VEL
LIN {X 0,Y 382.302,Z 975.679,A -85,B 0,C 180,E1 14794.658,E2 14794.658} C_VEL
LIN {X 0,Y 391.249,Z 954.249,A -85,B 0,C 180,E1 14792.774,E2 14792.774} C_VEL
LIN {X 0,Y 398.308,Z 935.434,A -85,B 0,C 180,E1 14791.403,E2 14791.403} C_VEL
LIN {X 0,Y 405.787,Z 912.924,A -85,B 0,C 180,E1 14790.036,E2 14790.036} C_VEL
LIN {X 0,Y 411.613,Z 892.272,A -85,B 0,C 180,E1 14789.012,E2 14789.012} C_VEL
LIN {X 0,Y 412.878,Z 887.506,A -85,B 0,C 180,E1 14788.8,E2 14788.8} C_VEL
LIN {X 0,Y 414.162,Z 880.462,A -85,B 0,C 180,E1 14788.383,E2 14788.383} C_VEL
LIN {X 0,Y 415.168,Z 861.941,A -85,B 0,C 180,E1 14786.958,E2 14786.958} C_VEL
LIN {X 0,Y 416.064,Z 855.712,A -85,B 0,C 180,E1 14786.664,E2 14786.664} C_VEL
LIN {X 0,Y 420.126,Z 830.814,A -85,B 0,C 180,E1 14786.016,E2 14786.016} C_VEL
LIN {X 0,Y 422.676,Z 808.458,A -85,B 0,C 180,E1 14785.582,E2 14785.582} C_VEL
LIN {X 0,Y 438.237,Z 612.268,A -85,B 0,C 180,E1 14782.437,E2 14782.437} C_VEL
LIN {X 0,Y 432.19,Z 601.97,A -85,B 0,C 180,E1 14780.094,E2 14780.094} C_VEL
LIN {X 0,Y 425.419,Z 591.266,A -85,B 0,C 180,E1 14777.085,E2 14777.085} C_VEL
LIN {X 0,Y 420.661,Z 584.036,A -85,B 0,C 180,E1 14774.593,E2 14774.593} C_VEL
LIN {X 0,Y 417.69,Z 579.611,A -85,B 0,C 180,E1 14772.793,E2 14772.793} C_VEL
LIN {X 0,Y 415.083,Z 575.644,A -85,B 0,C 180,E1 14770.971,E2 14770.971} C_VEL
LIN {X 0,Y 412.097,Z 571.096,A -85,B 0,C 180,E1 14768.441,E2 14768.441} C_VEL
LIN {X 0,Y 409.152,Z 567.12,A -85,B 0,C 180,E1 14765.047,E2 14765.047} C_VEL
LIN {X 0,Y 408.454,Z 565.52,A -85,B 0,C 180,E1 14763.79,E2 14763.79} C_VEL
LIN {X 0,Y 406.989,Z 564.529,A -85,B 0,C 180,E1 14758.311,E2 14758.311} C_VEL
LIN {X 0,Y 408.689,Z 565.834,A -85,B 0,C 180,E1 14753.256,E2 14753.256} C_VEL
LIN {X 0,Y 411.027,Z 570.01,A -85,B 0,C 180,E1 14750.054,E2 14750.054} C_VEL
LIN {X 0,Y 412.309,Z 571.493,A -85,B 0,C 180,E1 14748.813,E2 14748.813} C_VEL
LIN {X 0,Y 415.923,Z 576.903,A -85,B 0,C 180,E1 14745.877,E2 14745.877} C_VEL
LIN {X 0,Y 419.541,Z 582.308,A -85,B 0,C 180,E1 14743.524,E2 14743.524} C_VEL
LIN {X 0,Y 423.398,Z 589.083,A -85,B 0,C 180,E1 14741.337,E2 14741.337} C_VEL
LIN {X 0,Y 428.373,Z 598.04,A -85,B 0,C 180,E1 14738.897,E2 14738.897} C_VEL
LIN {X 0,Y 434.554,Z 609.875,A -85,B 0,C 180,E1 14736.255,E2 14736.255} C_VEL
LIN {X 0,Y 438.068,Z 617.207,A -85,B 0,C 180,E1 14734.883,E2 14734.883} C_VEL
LIN {X 0,Y 421.135,Z 829.72,A -85,B 0,C 180,E1 14731.46,E2 14731.46} C_VEL
LIN {X 0,Y 417.438,Z 856.576,A -85,B 0,C 180,E1 14730.897,E2 14730.897} C_VEL
LIN {X 0,Y 413.306,Z 877.949,A -85,B 0,C 180,E1 14730.319,E2 14730.319} C_VEL
LIN {X 0,Y 407.401,Z 902.388,A -85,B 0,C 180,E1 14729.466,E2 14729.466} C_VEL
LIN {X 0,Y 401.419,Z 922.923,A -85,B 0,C 180,E1 14728.554,E2 14728.554} C_VEL
LIN {X 0,Y 394.19,Z 944.789,A -85,B 0,C 180,E1 14727.367,E2 14727.367} C_VEL
LIN {X 0,Y 385.835,Z 966.585,A -85,B 0,C 180,E1 14725.893,E2 14725.893} C_VEL
LIN {X 0,Y 377.149,Z 987.138,A -85,B 0,C 180,E1 14724.22,E2 14724.22} C_VEL
LIN {X 0,Y 367.926,Z 1006.76,A -85,B 0,C 180,E1 14722.264,E2 14722.264} C_VEL
LIN {X 0,Y 359.167,Z 1024.127,A -85,B 0,C 180,E1 14720.207,E2 14720.207} C_VEL
LIN {X 0,Y 349.32,Z 1042.374,A -85,B 0,C 180,E1 14717.604,E2 14717.604} C_VEL
LIN {X 0,Y 340.714,Z 1057.528,A -85,B 0,C 180,E1 14715.013,E2 14715.013} C_VEL
LIN {X 0,Y 331.075,Z 1073.944,A -85,B 0,C 180,E1 14711.639,E2 14711.639} C_VEL
LIN {X 0,Y 323.342,Z 1086.824,A -85,B 0,C 180,E1 14708.431,E2 14708.431} C_VEL
LIN {X 0,Y 315.629,Z 1099.845,A -85,B 0,C 180,E1 14704.546,E2 14704.546} C_VEL
LIN {X 0,Y 309.514,Z 1110.379,A -85,B 0,C 180,E1 14700.692,E2 14700.692} C_VEL
LIN {X 0,Y 304.248,Z 1120.269,A -85,B 0,C 180,E1 14696.338,E2 14696.338} C_VEL
LIN {X 0,Y 300.299,Z 1128.48,A -85,B 0,C 180,E1 14691.724,E2 14691.724} C_VEL
LIN {X 0,Y 297.827,Z 1134.935,A -85,B 0,C 180,E1 14687.184,E2 14687.184} C_VEL
LIN {X 0,Y 296.46,Z 1139.806,A -85,B 0,C 180,E1 14682.466,E2 14682.466} C_VEL
LIN {X 0,Y 296.053,Z 1142.657,A -85,B 0,C 180,E1 14678.546,E2 14678.546} C_VEL
LIN {X 0,Y 296.01,Z 1144.478,A -85,B 0,C 180,E1 14674.456,E2 14674.456} C_VEL
LIN {X 0,Y 296.064,Z 1144.987,A -85,B 0,C 180,E1 14670.194,E2 14670.194} C_VEL
LIN {X 0,Y 296.038,Z 1144.23,A -85,B 0,C 180,E1 14666.321,E2 14666.321} C_VEL
LIN {X 0,Y 296.021,Z 1142.594,A -85,B 0,C 180,E1 14662.821,E2 14662.821} C_VEL
LIN {X 0,Y 296.237,Z 1139.861,A -85,B 0,C 180,E1 14659.105,E2 14659.105} C_VEL
LIN {X 0,Y 297.198,Z 1134.935,A -85,B 0,C 180,E1 14654.386,E2 14654.386} C_VEL
LIN {X 0,Y 299.049,Z 1128.767,A -85,B 0,C 180,E1 14650.059,E2 14650.059} C_VEL
LIN {X 0,Y 302.031,Z 1121.174,A -85,B 0,C 180,E1 14645.763,E2 14645.763} C_VEL
LIN {X 0,Y 306.484,Z 1111.365,A -85,B 0,C 180,E1 14641.342,E2 14641.342} C_VEL
LIN {X 0,Y 311.542,Z 1101.288,A -85,B 0,C 180,E1 14637.576,E2 14637.576} C_VEL
LIN {X 0,Y 318.7,Z 1087.737,A -85,B 0,C 180,E1 14633.408,E2 14633.408} C_VEL
LIN {X 0,Y 325.547,Z 1075.037,A -85,B 0,C 180,E1 14630.162,E2 14630.162} C_VEL
LIN {X 0,Y 334.606,Z 1058.156,A -85,B 0,C 180,E1 14626.583,E2 14626.583} C_VEL
LIN {X 0,Y 342.63,Z 1042.798,A -85,B 0,C 180,E1 14623.878,E2 14623.878} C_VEL
LIN {X 0,Y 352.127,Z 1023.764,A -85,B 0,C 180,E1 14621.084,E2 14621.084} C_VEL
LIN {X 0,Y 360.182,Z 1006.592,A -85,B 0,C 180,E1 14618.986,E2 14618.986} C_VEL
LIN {X 0,Y 369.245,Z 985.781,A -85,B 0,C 180,E1 14616.854,E2 14616.854} C_VEL
LIN {X 0,Y 376.777,Z 966.81,A -85,B 0,C 180,E1 14615.251,E2 14615.251} C_VEL
LIN {X 0,Y 384.643,Z 945.042,A -85,B 0,C 180,E1 14613.71,E2 14613.71} C_VEL
LIN {X 0,Y 391.248,Z 923.935,A -85,B 0,C 180,E1 14612.503,E2 14612.503} C_VEL
LIN {X 0,Y 396.915,Z 903.437,A -85,B 0,C 180,E1 14611.535,E2 14611.535} C_VEL
LIN {X 0,Y 402.665,Z 878.523,A -85,B 0,C 180,E1 14610.612,E2 14610.612} C_VEL
LIN {X 0,Y 406.669,Z 856.8,A -85,B 0,C 180,E1 14609.992,E2 14609.992} C_VEL
LIN {X 0,Y 410.186,Z 829.721,A -85,B 0,C 180,E1 14609.402,E2 14609.402} C_VEL
LIN {X 0,Y 426.327,Z 613.763,A -85,B 0,C 180,E1 14605.846,E2 14605.846} C_VEL
LIN {X 0,Y 426.584,Z 609.227,A -85,B 0,C 180,E1 14605.751,E2 14605.751} C_VEL
LIN {X 0,Y 419.267,Z 594.499,A -85,B 0,C 180,E1 14603.173,E2 14603.173} C_VEL
LIN {X 0,Y 412.272,Z 581.583,A -85,B 0,C 180,E1 14600.404,E2 14600.404} C_VEL
LIN {X 0,Y 406.439,Z 571.459,A -85,B 0,C 180,E1 14597.762,E2 14597.762} C_VEL
LIN {X 0,Y 401.495,Z 564.334,A -85,B 0,C 180,E1 14595.233,E2 14595.233} C_VEL
LIN {X 0,Y 398.537,Z 560.1,A -85,B 0,C 180,E1 14593.493,E2 14593.493} C_VEL
LIN {X 0,Y 395.213,Z 555.333,A -85,B 0,C 180,E1 14591.234,E2 14591.234} C_VEL
LIN {X 0,Y 392.107,Z 550.888,A -85,B 0,C 180,E1 14588.653,E2 14588.653} C_VEL
LIN {X 0,Y 388.603,Z 546.231,A -85,B 0,C 180,E1 14584.575,E2 14584.575} C_VEL
LIN {X 0,Y 388.063,Z 544.851,A -85,B 0,C 180,E1 14583.545,E2 14583.545} C_VEL
LIN {X 0,Y 386.554,Z 543.995,A -85,B 0,C 180,E1 14577.331,E2 14577.331} C_VEL
LIN {X 0,Y 388.193,Z 545.058,A -85,B 0,C 180,E1 14572.675,E2 14572.675} C_VEL
LIN {X 0,Y 390.1,Z 548.839,A -85,B 0,C 180,E1 14569.813,E2 14569.813} C_VEL
LIN {X 0,Y 392.13,Z 550.974,A -85,B 0,C 180,E1 14567.781,E2 14567.781} C_VEL
LIN {X 0,Y 395.251,Z 555.419,A -85,B 0,C 180,E1 14565.196,E2 14565.196} C_VEL
LIN {X 0,Y 399.865,Z 561.982,A -85,B 0,C 180,E1 14562.162,E2 14562.162} C_VEL
LIN {X 0,Y 403.691,Z 567.58,A -85,B 0,C 180,E1 14560.051,E2 14560.051} C_VEL
LIN {X 0,Y 408.856,Z 575.096,A -85,B 0,C 180,E1 14557.583,E2 14557.583} C_VEL
LIN {X 0,Y 416.677,Z 587.235,A -85,B 0,C 180,E1 14554.371,E2 14554.371} C_VEL
LIN {X 0,Y 424.779,Z 600.813,A -85,B 0,C 180,E1 14551.494,E2 14551.494} C_VEL
LIN {X 0,Y 426.867,Z 604.646,A -85,B 0,C 180,E1 14550.802,E2 14550.802} C_VEL
LIN {X 0,Y 410.951,Z 815.616,A -85,B 0,C 180,E1 14547.345,E2 14547.345} C_VEL
LIN {X 0,Y 407.541,Z 842.184,A -85,B 0,C 180,E1 14546.739,E2 14546.739} C_VEL
LIN {X 0,Y 403.848,Z 863.241,A -85,B 0,C 180,E1 14546.088,E2 14546.088} C_VEL
LIN {X 0,Y 398.509,Z 887.508,A -85,B 0,C 180,E1 14545.132,E2 14545.132} C_VEL
LIN {X 0,Y 393.046,Z 907.957,A -85,B 0,C 180,E1 14544.121,E2 14544.121} C_VEL
LIN {X 0,Y 386.136,Z 930.515,A -85,B 0,C 180,E1 14542.77,E2 14542.77} C_VEL
LIN {X 0,Y 378.91,Z 950.722,A -85,B 0,C 180,E1 14541.287,E2 14541.287} C_VEL
LIN {X 0,Y 371.152,Z 970.526,A -85,B 0,C 180,E1 14539.558,E2 14539.558} C_VEL
LIN {X 0,Y 362.405,Z 990.525,A -85,B 0,C 180,E1 14537.448,E2 14537.448} C_VEL
LIN {X 0,Y 354.389,Z 1007.549,A -85,B 0,C 180,E1 14535.317,E2 14535.317} C_VEL
LIN {X 0,Y 345.376,Z 1025.388,A -85,B 0,C 180,E1 14532.645,E2 14532.645} C_VEL
LIN {X 0,Y 337.506,Z 1040.16,A -85,B 0,C 180,E1 14530.007,E2 14530.007} C_VEL
LIN {X 0,Y 328.689,Z 1056.116,A -85,B 0,C 180,E1 14526.601,E2 14526.601} C_VEL
LIN {X 0,Y 321.643,Z 1068.59,A -85,B 0,C 180,E1 14523.384,E2 14523.384} C_VEL
LIN {X 0,Y 314.608,Z 1081.155,A -85,B 0,C 180,E1 14519.513,E2 14519.513} C_VEL
LIN {X 0,Y 309.021,Z 1091.264,A -85,B 0,C 180,E1 14515.695,E2 14515.695} C_VEL
LIN {X 0,Y 304.192,Z 1100.711,A -85,B 0,C 180,E1 14511.399,E2 14511.399} C_VEL
LIN {X 0,Y 300.635,Z 1108.255,A -85,B 0,C 180,E1 14507.019,E2 14507.019} C_VEL
LIN {X 0,Y 298.334,Z 1114.1,A -85,B 0,C 180,E1 14502.78,E2 14502.78} C_VEL
LIN {X 0,Y 296.839,Z 1118.988,A -85,B 0,C 180,E1 14497.938,E2 14497.938} C_VEL
LIN {X 0,Y 296.281,Z 1121.677,A -85,B 0,C 180,E1 14494.064,E2 14494.064} C_VEL
LIN {X 0,Y 296.119,Z 1123.332,A -85,B 0,C 180,E1 14490.193,E2 14490.193} C_VEL
LIN {X 0,Y 296.067,Z 1123.943,A -85,B 0,C 180,E1 14485.739,E2 14485.739} C_VEL
LIN {X 0,Y 296.216,Z 1123.215,A -85,B 0,C 180,E1 14481.654,E2 14481.654} C_VEL
LIN {X 0,Y 296.597,Z 1121.478,A -85,B 0,C 180,E1 14477.738,E2 14477.738} C_VEL
LIN {X 0,Y 297.773,Z 1118.01,A -85,B 0,C 180,E1 14473.014,E2 14473.014} C_VEL
LIN {X 0,Y 299.772,Z 1113.262,A -85,B 0,C 180,E1 14468.68,E2 14468.68} C_VEL
LIN {X 0,Y 302.71,Z 1107.472,A -85,B 0,C 180,E1 14464.57,E2 14464.57} C_VEL
LIN {X 0,Y 307.515,Z 1098.954,A -85,B 0,C 180,E1 14459.872,E2 14459.872} C_VEL
LIN {X 0,Y 312.854,Z 1090.169,A -85,B 0,C 180,E1 14455.992,E2 14455.992} C_VEL
LIN {X 0,Y 320.507,Z 1077.943,A -85,B 0,C 180,E1 14451.623,E2 14451.623} C_VEL
LIN {X 0,Y 327.682,Z 1066.573,A -85,B 0,C 180,E1 14448.302,E2 14448.302} C_VEL
LIN {X 0,Y 337.15,Z 1051.287,A -85,B 0,C 180,E1 14444.62,E2 14444.62} C_VEL
LIN {X 0,Y 345.301,Z 1037.661,A -85,B 0,C 180,E1 14441.91,E2 14441.91} C_VEL
LIN {X 0,Y 355.225,Z 1020.309,A -85,B 0,C 180,E1 14439.023,E2 14439.023} C_VEL
LIN {X 0,Y 363.74,Z 1004.337,A -85,B 0,C 180,E1 14436.817,E2 14436.817} C_VEL
LIN {X 0,Y 373.227,Z 985.394,A -85,B 0,C 180,E1 14434.608,E2 14434.608} C_VEL
LIN {X 0,Y 382.08,Z 965.662,A -85,B 0,C 180,E1 14432.716,E2 14432.716} C_VEL
LIN {X 0,Y 390.481,Z 945.209,A -85,B 0,C 180,E1 14431.069,E2 14431.069} C_VEL
LIN {X 0,Y 398.238,Z 923.472,A -85,B 0,C 180,E1 14429.645,E2 14429.645} C_VEL
LIN {X 0,Y 405.172,Z 901.395,A -85,B 0,C 180,E1 14428.443,E2 14428.443} C_VEL
LIN {X 0,Y 411.211,Z 878.138,A -85,B 0,C 180,E1 14427.436,E2 14427.436} C_VEL
LIN {X 0,Y 415.97,Z 856.175,A -85,B 0,C 180,E1 14426.679,E2 14426.679} C_VEL
LIN {X 0,Y 416.064,Z 855.712,A -85,B 0,C 180,E1 14426.664,E2 14426.664} C_VEL
LIN {X 0,Y 416.98,Z 848.403,A -85,B 0,C 180,E1 14426.323,E2 14426.323} C_VEL
LIN {X 0,Y 417.028,Z 830.211,A -85,B 0,C 180,E1 14425.141,E2 14425.141} C_VEL
LIN {X 0,Y 417.621,Z 822.757,A -85,B 0,C 180,E1 14424.861,E2 14424.861} C_VEL
LIN {X 0,Y 420.985,Z 785.72,A -85,B 0,C 180,E1 14424.233,E2 14424.233} C_VEL
LIN {X 0,Y 434.641,Z 616.956,A -85,B 0,C 180,E1 14421.534,E2 14421.534} C_VEL
LIN {X 0,Y 428.972,Z 607.313,A -85,B 0,C 180,E1 14419.223,E2 14419.223} C_VEL
LIN {X 0,Y 422.723,Z 597.088,A -85,B 0,C 180,E1 14416.278,E2 14416.278} C_VEL
LIN {X 0,Y 417.027,Z 588.232,A -85,B 0,C 180,E1 14413.025,E2 14413.025} C_VEL
LIN {X 0,Y 413.55,Z 583.145,A -85,B 0,C 180,E1 14410.589,E2 14410.589} C_VEL
LIN {X 0,Y 410.607,Z 578.591,A -85,B 0,C 180,E1 14407.979,E2 14407.979} C_VEL
LIN {X 0,Y 407.994,Z 574.816,A -85,B 0,C 180,E1 14404.78,E2 14404.78} C_VEL
LIN {X 0,Y 407.397,Z 573.427,A -85,B 0,C 180,E1 14403.659,E2 14403.659} C_VEL
LIN {X 0,Y 406.014,Z 572.47,A -85,B 0,C 180,E1 14398.307,E2 14398.307} C_VEL
LIN {X 0,Y 407.595,Z 573.645,A -85,B 0,C 180,E1 14393.45,E2 14393.45} C_VEL
LIN {X 0,Y 409.791,Z 577.75,A -85,B 0,C 180,E1 14390.307,E2 14390.307} C_VEL
LIN {X 0,Y 411.106,Z 579.335,A -85,B 0,C 180,E1 14388.993,E2 14388.993} C_VEL
LIN {X 0,Y 414.561,Z 584.615,A -85,B 0,C 180,E1 14386.114,E2 14386.114} C_VEL
LIN {X 0,Y 418.107,Z 590.037,A -85,B 0,C 180,E1 14383.752,E2 14383.752} C_VEL
LIN {X 0,Y 422.789,Z 598.394,A -85,B 0,C 180,E1 14381.085,E2 14381.085} C_VEL
LIN {X 0,Y 428.046,Z 608.406,A -85,B 0,C 180,E1 14378.521,E2 14378.521} C_VEL
LIN {X 0,Y 433.57,Z 619.484,A -85,B 0,C 180,E1 14376.161,E2 14376.161} C_VEL
LIN {X 0,Y 434.5,Z 621.7,A -85,B 0,C 180,E1 14375.778,E2 14375.778} C_VEL
LIN {X 0,Y 417.511,Z 829.632,A -85,B 0,C 180,E1 14372.439,E2 14372.439} C_VEL
LIN {X 0,Y 413.736,Z 856.44,A -85,B 0,C 180,E1 14371.88,E2 14371.88} C_VEL
LIN {X 0,Y 409.543,Z 877.711,A -85,B 0,C 180,E1 14371.309,E2 14371.309} C_VEL
LIN {X 0,Y 403.428,Z 902.462,A -85,B 0,C 180,E1 14370.453,E2 14370.453} C_VEL
LIN {X 0,Y 397.283,Z 923.079,A -85,B 0,C 180,E1 14369.544,E2 14369.544} C_VEL
LIN {X 0,Y 389.55,Z 945.797,A -85,B 0,C 180,E1 14368.309,E2 14368.309} C_VEL
LIN {X 0,Y 381.352,Z 966.615,A -85,B 0,C 180,E1 14366.9,E2 14366.9} C_VEL
LIN {X 0,Y 372.454,Z 987.138,A -85,B 0,C 180,E1 14365.234,E2 14365.234} C_VEL
LIN {X 0,Y 362.987,Z 1006.709,A -85,B 0,C 180,E1 14363.283,E2 14363.283} C_VEL
LIN {X 0,Y 353.981,Z 1024.054,A -85,B 0,C 180,E1 14361.226,E2 14361.226} C_VEL
LIN {X 0,Y 343.827,Z 1042.262,A -85,B 0,C 180,E1 14358.616,E2 14358.616} C_VEL
LIN {X 0,Y 334.933,Z 1057.401,A -85,B 0,C 180,E1 14356.011,E2 14356.011} C_VEL
LIN {X 0,Y 324.943,Z 1073.787,A -85,B 0,C 180,E1 14352.607,E2 14352.607} C_VEL
LIN {X 0,Y 316.895,Z 1086.654,A -85,B 0,C 180,E1 14349.362,E2 14349.362} C_VEL
LIN {X 0,Y 308.832,Z 1099.65,A -85,B 0,C 180,E1 14345.418,E2 14345.418} C_VEL
LIN {X 0,Y 302.317,Z 1110.34,A -85,B 0,C 180,E1 14341.425,E2 14341.425} C_VEL
LIN {X 0,Y 296.859,Z 1120.047,A -85,B 0,C 180,E1 14337.047,E2 14337.047} C_VEL
LIN {X 0,Y 292.778,Z 1127.984,A -85,B 0,C 180,E1 14332.489,E2 14332.489} C_VEL
LIN {X 0,Y 290.146,Z 1134.276,A -85,B 0,C 180,E1 14327.983,E2 14327.983} C_VEL
LIN {X 0,Y 288.562,Z 1139.38,A -85,B 0,C 180,E1 14323.016,E2 14323.016} C_VEL
LIN {X 0,Y 288.075,Z 1142.272,A -85,B 0,C 180,E1 14318.986,E2 14318.986} C_VEL
LIN {X 0,Y 287.996,Z 1144.062,A -85,B 0,C 180,E1 14314.979,E2 14314.979} C_VEL
LIN {X 0,Y 288.057,Z 1144.761,A -85,B 0,C 180,E1 14310.796,E2 14310.796} C_VEL
LIN {X 0,Y 288.04,Z 1144.072,A -85,B 0,C 180,E1 14306.617,E2 14306.617} C_VEL
LIN {X 0,Y 288.024,Z 1142.403,A -85,B 0,C 180,E1 14302.821,E2 14302.821} C_VEL
LIN {X 0,Y 288.271,Z 1139.543,A -85,B 0,C 180,E1 14298.8,E2 14298.8} C_VEL
LIN {X 0,Y 289.343,Z 1134.509,A -85,B 0,C 180,E1 14293.883,E2 14293.883} C_VEL
